// TIA Portal V17 export
// export: Created 2025-03-05T08:01:27.4239507Z, ExportSetting WithDefaults, DisplayName Totally Integrated Automation Portal, DisplayVersion V17 Update 8, DisplayName TIA Portal Openness, DisplayVersion V17 Update 8, DisplayName TIA Portal Version Control Interface, DisplayVersion V17, DisplayName SINAMICS Startdrive Advanced, DisplayVersion V17 SP2, DisplayName SINAMICS Startdrive G110M, G120, G120C, G120D, G120P, G115D, DisplayVersion V17 SP2, DisplayName SINAMICS Startdrive G130, G150, S120, S150, SINAMICS MV, S210, DisplayVersion V17 SP2, DisplayName STEP 7 Professional, DisplayVersion V17 Update 8, DisplayName SINUMERIK ONE STEP 7 Toolbox, DisplayVersion V17 Update 12, DisplayName SINUMERIK 840D sl STEP 7 Toolbox, DisplayVersion V17 Update 12, DisplayName STEP 7 Safety, DisplayVersion V17 Update 6, DisplayName WinCC Advanced, DisplayVersion V17 Update 8
FUNCTION "FC16013_METHOD_CALLS_U02_STA2_MEAS" : Void   // FC16013, LAD
{ S7_Optimized_Access := 'TRUE' }
VERSION : 0.1
// stored: AutoNumber false, IsIECCheckEnabled false, SetENOAutomatically false, UDAEnableTagReadback false
   VAR_TEMP
      AUX_WSTRING_PART_ID_STA2 : WString;
      AUX_WCHARS : Array[0..63] of WChar;
      index : Int;
      ALARM_AUX : Bool;
   END_VAR
   VAR_TEMP   // added for the SCL form of the ladder/FBD networks
      _w1 : Bool;
      _w2 : Bool;
   END_VAR
BEGIN

REGION Network 1 (SCL): TRANSFORM TO WCHARS
   FOR #index := 0 TO 63 DO
       #AUX_WCHARS[#index] := CHAR_TO_WCHAR("DB8000_PART_STATUS".UNIT_02.STATION_2.PART_A.PART_ID[#index]);
   END_FOR;
END_REGION

REGION Network 2: TRANSFORM TO WSTRING
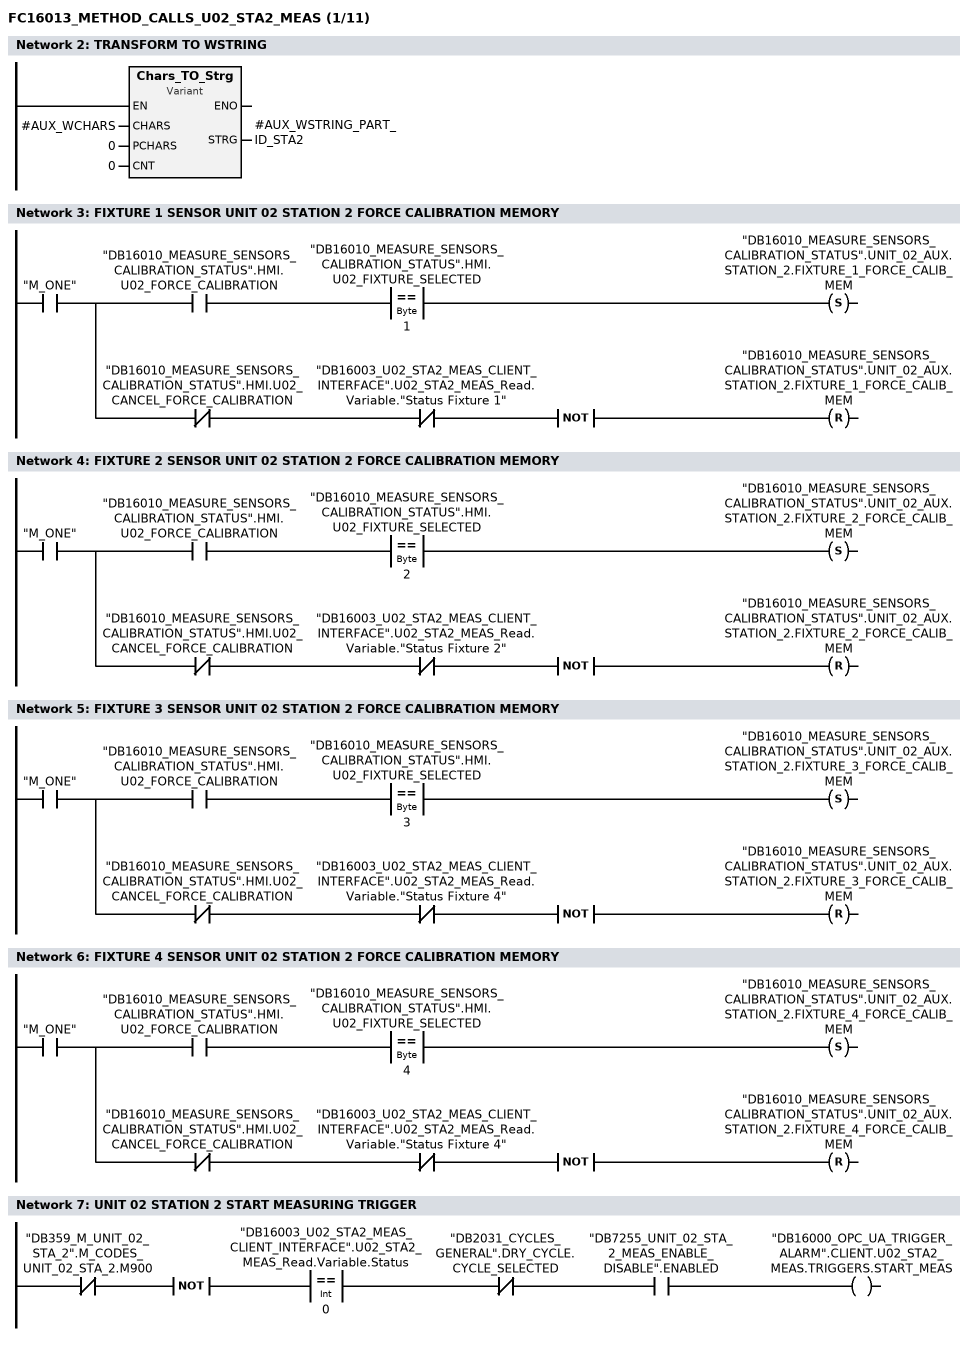
   RUNG wire#powerrail
      { S7_Templates := "[ptr_type := Variant, str_type := WString]" } Chars_TO_Strg(Chars := #AUX_WCHARS, pChars := 0, Cnt := 0, Strg => #AUX_WSTRING_PART_ID_STA2)
   END_RUNG
   // the same network as SCL:
   Chars_TO_Strg(Chars := #AUX_WCHARS, pChars := 0, Cnt := 0, Strg => #AUX_WSTRING_PART_ID_STA2);
END_REGION

REGION Network 3: FIXTURE 1 SENSOR UNIT 02 STATION 2 FORCE CALIBRATION MEMORY
   RUNG wire#powerrail
      Contact( "M_ONE" )
      wire#w1
      Contact( "DB16010_MEASURE_SENSORS_CALIBRATION_STATUS".HMI.U02_FORCE_CALIBRATION )
      { S7_Templates := "SrcType := Byte" } EQ_Contact(in1 := "DB16010_MEASURE_SENSORS_CALIBRATION_STATUS".HMI.U02_FIXTURE_SELECTED, in2 := 1)
      S_Coil( "DB16010_MEASURE_SENSORS_CALIBRATION_STATUS".UNIT_02_AUX.STATION_2.FIXTURE_1_FORCE_CALIB_MEM )
   END_RUNG
   RUNG wire#w1
      I_Contact( "DB16010_MEASURE_SENSORS_CALIBRATION_STATUS".HMI.U02_CANCEL_FORCE_CALIBRATION )
      I_Contact( "DB16003_U02_STA2_MEAS_CLIENT_INTERFACE".U02_STA2_MEAS_Read.Variable."Status Fixture 1" )
      Not()
      R_Coil( "DB16010_MEASURE_SENSORS_CALIBRATION_STATUS".UNIT_02_AUX.STATION_2.FIXTURE_1_FORCE_CALIB_MEM )
   END_RUNG
   // the same network as SCL:
   IF "M_ONE" AND "DB16010_MEASURE_SENSORS_CALIBRATION_STATUS".HMI.U02_FORCE_CALIBRATION AND ("DB16010_MEASURE_SENSORS_CALIBRATION_STATUS".HMI.U02_FIXTURE_SELECTED = 1) THEN
       "DB16010_MEASURE_SENSORS_CALIBRATION_STATUS".UNIT_02_AUX.STATION_2.FIXTURE_1_FORCE_CALIB_MEM := TRUE;
   END_IF;
   IF NOT ("M_ONE" AND NOT "DB16010_MEASURE_SENSORS_CALIBRATION_STATUS".HMI.U02_CANCEL_FORCE_CALIBRATION AND NOT "DB16003_U02_STA2_MEAS_CLIENT_INTERFACE".U02_STA2_MEAS_Read.Variable."Status Fixture 1") THEN
       "DB16010_MEASURE_SENSORS_CALIBRATION_STATUS".UNIT_02_AUX.STATION_2.FIXTURE_1_FORCE_CALIB_MEM := FALSE;
   END_IF;
END_REGION

REGION Network 4: FIXTURE 2 SENSOR UNIT 02 STATION 2 FORCE CALIBRATION MEMORY
   RUNG wire#powerrail
      Contact( "M_ONE" )
      wire#w1
      Contact( "DB16010_MEASURE_SENSORS_CALIBRATION_STATUS".HMI.U02_FORCE_CALIBRATION )
      { S7_Templates := "SrcType := Byte" } EQ_Contact(in1 := "DB16010_MEASURE_SENSORS_CALIBRATION_STATUS".HMI.U02_FIXTURE_SELECTED, in2 := 2)
      S_Coil( "DB16010_MEASURE_SENSORS_CALIBRATION_STATUS".UNIT_02_AUX.STATION_2.FIXTURE_2_FORCE_CALIB_MEM )
   END_RUNG
   RUNG wire#w1
      I_Contact( "DB16010_MEASURE_SENSORS_CALIBRATION_STATUS".HMI.U02_CANCEL_FORCE_CALIBRATION )
      I_Contact( "DB16003_U02_STA2_MEAS_CLIENT_INTERFACE".U02_STA2_MEAS_Read.Variable."Status Fixture 2" )
      Not()
      R_Coil( "DB16010_MEASURE_SENSORS_CALIBRATION_STATUS".UNIT_02_AUX.STATION_2.FIXTURE_2_FORCE_CALIB_MEM )
   END_RUNG
   // the same network as SCL:
   IF "M_ONE" AND "DB16010_MEASURE_SENSORS_CALIBRATION_STATUS".HMI.U02_FORCE_CALIBRATION AND ("DB16010_MEASURE_SENSORS_CALIBRATION_STATUS".HMI.U02_FIXTURE_SELECTED = 2) THEN
       "DB16010_MEASURE_SENSORS_CALIBRATION_STATUS".UNIT_02_AUX.STATION_2.FIXTURE_2_FORCE_CALIB_MEM := TRUE;
   END_IF;
   IF NOT ("M_ONE" AND NOT "DB16010_MEASURE_SENSORS_CALIBRATION_STATUS".HMI.U02_CANCEL_FORCE_CALIBRATION AND NOT "DB16003_U02_STA2_MEAS_CLIENT_INTERFACE".U02_STA2_MEAS_Read.Variable."Status Fixture 2") THEN
       "DB16010_MEASURE_SENSORS_CALIBRATION_STATUS".UNIT_02_AUX.STATION_2.FIXTURE_2_FORCE_CALIB_MEM := FALSE;
   END_IF;
END_REGION

REGION Network 5: FIXTURE 3 SENSOR UNIT 02 STATION 2 FORCE CALIBRATION MEMORY
   RUNG wire#powerrail
      Contact( "M_ONE" )
      wire#w1
      Contact( "DB16010_MEASURE_SENSORS_CALIBRATION_STATUS".HMI.U02_FORCE_CALIBRATION )
      { S7_Templates := "SrcType := Byte" } EQ_Contact(in1 := "DB16010_MEASURE_SENSORS_CALIBRATION_STATUS".HMI.U02_FIXTURE_SELECTED, in2 := 3)
      S_Coil( "DB16010_MEASURE_SENSORS_CALIBRATION_STATUS".UNIT_02_AUX.STATION_2.FIXTURE_3_FORCE_CALIB_MEM )
   END_RUNG
   RUNG wire#w1
      I_Contact( "DB16010_MEASURE_SENSORS_CALIBRATION_STATUS".HMI.U02_CANCEL_FORCE_CALIBRATION )
      I_Contact( "DB16003_U02_STA2_MEAS_CLIENT_INTERFACE".U02_STA2_MEAS_Read.Variable."Status Fixture 4" )
      Not()
      R_Coil( "DB16010_MEASURE_SENSORS_CALIBRATION_STATUS".UNIT_02_AUX.STATION_2.FIXTURE_3_FORCE_CALIB_MEM )
   END_RUNG
   // the same network as SCL:
   IF "M_ONE" AND "DB16010_MEASURE_SENSORS_CALIBRATION_STATUS".HMI.U02_FORCE_CALIBRATION AND ("DB16010_MEASURE_SENSORS_CALIBRATION_STATUS".HMI.U02_FIXTURE_SELECTED = 3) THEN
       "DB16010_MEASURE_SENSORS_CALIBRATION_STATUS".UNIT_02_AUX.STATION_2.FIXTURE_3_FORCE_CALIB_MEM := TRUE;
   END_IF;
   IF NOT ("M_ONE" AND NOT "DB16010_MEASURE_SENSORS_CALIBRATION_STATUS".HMI.U02_CANCEL_FORCE_CALIBRATION AND NOT "DB16003_U02_STA2_MEAS_CLIENT_INTERFACE".U02_STA2_MEAS_Read.Variable."Status Fixture 4") THEN
       "DB16010_MEASURE_SENSORS_CALIBRATION_STATUS".UNIT_02_AUX.STATION_2.FIXTURE_3_FORCE_CALIB_MEM := FALSE;
   END_IF;
END_REGION

REGION Network 6: FIXTURE 4 SENSOR UNIT 02 STATION 2 FORCE CALIBRATION MEMORY
   RUNG wire#powerrail
      Contact( "M_ONE" )
      wire#w1
      Contact( "DB16010_MEASURE_SENSORS_CALIBRATION_STATUS".HMI.U02_FORCE_CALIBRATION )
      { S7_Templates := "SrcType := Byte" } EQ_Contact(in1 := "DB16010_MEASURE_SENSORS_CALIBRATION_STATUS".HMI.U02_FIXTURE_SELECTED, in2 := 4)
      S_Coil( "DB16010_MEASURE_SENSORS_CALIBRATION_STATUS".UNIT_02_AUX.STATION_2.FIXTURE_4_FORCE_CALIB_MEM )
   END_RUNG
   RUNG wire#w1
      I_Contact( "DB16010_MEASURE_SENSORS_CALIBRATION_STATUS".HMI.U02_CANCEL_FORCE_CALIBRATION )
      I_Contact( "DB16003_U02_STA2_MEAS_CLIENT_INTERFACE".U02_STA2_MEAS_Read.Variable."Status Fixture 4" )
      Not()
      R_Coil( "DB16010_MEASURE_SENSORS_CALIBRATION_STATUS".UNIT_02_AUX.STATION_2.FIXTURE_4_FORCE_CALIB_MEM )
   END_RUNG
   // the same network as SCL:
   IF "M_ONE" AND "DB16010_MEASURE_SENSORS_CALIBRATION_STATUS".HMI.U02_FORCE_CALIBRATION AND ("DB16010_MEASURE_SENSORS_CALIBRATION_STATUS".HMI.U02_FIXTURE_SELECTED = 4) THEN
       "DB16010_MEASURE_SENSORS_CALIBRATION_STATUS".UNIT_02_AUX.STATION_2.FIXTURE_4_FORCE_CALIB_MEM := TRUE;
   END_IF;
   IF NOT ("M_ONE" AND NOT "DB16010_MEASURE_SENSORS_CALIBRATION_STATUS".HMI.U02_CANCEL_FORCE_CALIBRATION AND NOT "DB16003_U02_STA2_MEAS_CLIENT_INTERFACE".U02_STA2_MEAS_Read.Variable."Status Fixture 4") THEN
       "DB16010_MEASURE_SENSORS_CALIBRATION_STATUS".UNIT_02_AUX.STATION_2.FIXTURE_4_FORCE_CALIB_MEM := FALSE;
   END_IF;
END_REGION

REGION Network 7: UNIT 02 STATION 2 START MEASURING TRIGGER
   RUNG wire#powerrail
      I_Contact( "DB359_M_UNIT_02_STA_2".M_CODES_UNIT_02_STA_2.M900 )
      Not()
      { S7_Templates := "SrcType := Int" } EQ_Contact(in1 := "DB16003_U02_STA2_MEAS_CLIENT_INTERFACE".U02_STA2_MEAS_Read.Variable.Status, in2 := 0)
      I_Contact( "DB2031_CYCLES_GENERAL".DRY_CYCLE.CYCLE_SELECTED )
      Contact( "DB7255_UNIT_02_STA_2_MEAS_ENABLE_DISABLE".ENABLED )
      Coil( "DB16000_OPC_UA_TRIGGER_ALARM".CLIENT.U02_STA2_MEAS.TRIGGERS.START_MEAS )
   END_RUNG
   // the same network as SCL:
   "DB16000_OPC_UA_TRIGGER_ALARM".CLIENT.U02_STA2_MEAS.TRIGGERS.START_MEAS := NOT (NOT "DB359_M_UNIT_02_STA_2".M_CODES_UNIT_02_STA_2.M900) AND ("DB16003_U02_STA2_MEAS_CLIENT_INTERFACE".U02_STA2_MEAS_Read.Variable.Status = 0) AND NOT "DB2031_CYCLES_GENERAL".DRY_CYCLE.CYCLE_SELECTED AND "DB7255_UNIT_02_STA_2_MEAS_ENABLE_DISABLE".ENABLED;
END_REGION

REGION Network 8: UNIT 02 STATION 2 START CALIBRATING TRIGGER
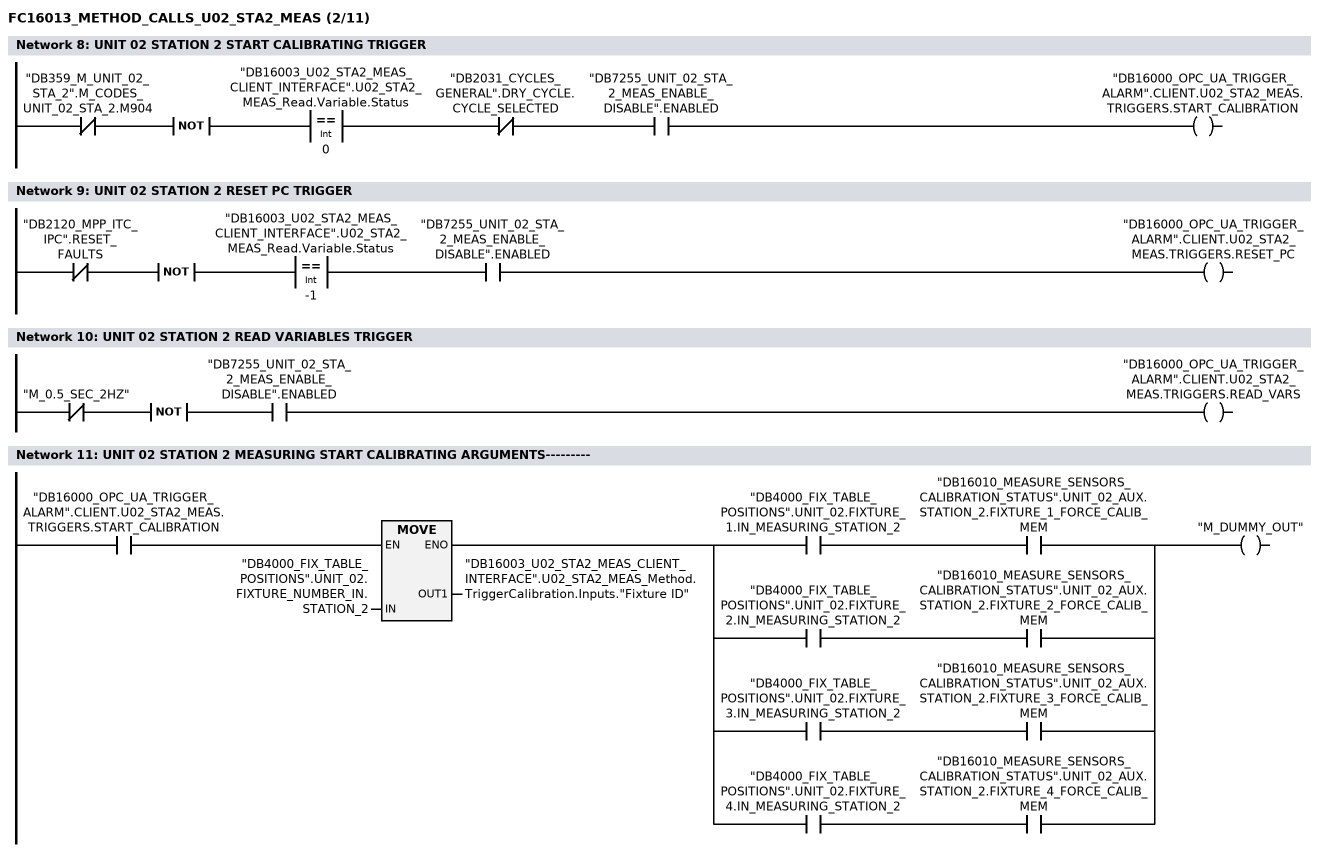
   RUNG wire#powerrail
      I_Contact( "DB359_M_UNIT_02_STA_2".M_CODES_UNIT_02_STA_2.M904 )
      Not()
      { S7_Templates := "SrcType := Int" } EQ_Contact(in1 := "DB16003_U02_STA2_MEAS_CLIENT_INTERFACE".U02_STA2_MEAS_Read.Variable.Status, in2 := 0)
      I_Contact( "DB2031_CYCLES_GENERAL".DRY_CYCLE.CYCLE_SELECTED )
      Contact( "DB7255_UNIT_02_STA_2_MEAS_ENABLE_DISABLE".ENABLED )
      Coil( "DB16000_OPC_UA_TRIGGER_ALARM".CLIENT.U02_STA2_MEAS.TRIGGERS.START_CALIBRATION )
   END_RUNG
   // the same network as SCL:
   "DB16000_OPC_UA_TRIGGER_ALARM".CLIENT.U02_STA2_MEAS.TRIGGERS.START_CALIBRATION := NOT (NOT "DB359_M_UNIT_02_STA_2".M_CODES_UNIT_02_STA_2.M904) AND ("DB16003_U02_STA2_MEAS_CLIENT_INTERFACE".U02_STA2_MEAS_Read.Variable.Status = 0) AND NOT "DB2031_CYCLES_GENERAL".DRY_CYCLE.CYCLE_SELECTED AND "DB7255_UNIT_02_STA_2_MEAS_ENABLE_DISABLE".ENABLED;
END_REGION

REGION Network 9: UNIT 02 STATION 2 RESET PC TRIGGER
   RUNG wire#powerrail
      I_Contact( "DB2120_MPP_ITC_IPC".RESET_FAULTS )
      Not()
      { S7_Templates := "SrcType := Int" } EQ_Contact(in1 := "DB16003_U02_STA2_MEAS_CLIENT_INTERFACE".U02_STA2_MEAS_Read.Variable.Status, in2 := -1)
      Contact( "DB7255_UNIT_02_STA_2_MEAS_ENABLE_DISABLE".ENABLED )
      Coil( "DB16000_OPC_UA_TRIGGER_ALARM".CLIENT.U02_STA2_MEAS.TRIGGERS.RESET_PC )
   END_RUNG
   // the same network as SCL:
   "DB16000_OPC_UA_TRIGGER_ALARM".CLIENT.U02_STA2_MEAS.TRIGGERS.RESET_PC := NOT (NOT "DB2120_MPP_ITC_IPC".RESET_FAULTS) AND ("DB16003_U02_STA2_MEAS_CLIENT_INTERFACE".U02_STA2_MEAS_Read.Variable.Status = (-1)) AND "DB7255_UNIT_02_STA_2_MEAS_ENABLE_DISABLE".ENABLED;
END_REGION

REGION Network 10: UNIT 02 STATION 2 READ VARIABLES TRIGGER
   RUNG wire#powerrail
      I_Contact( "M_0.5_SEC_2HZ" )
      Not()
      Contact( "DB7255_UNIT_02_STA_2_MEAS_ENABLE_DISABLE".ENABLED )
      Coil( "DB16000_OPC_UA_TRIGGER_ALARM".CLIENT.U02_STA2_MEAS.TRIGGERS.READ_VARS )
   END_RUNG
   // the same network as SCL:
   "DB16000_OPC_UA_TRIGGER_ALARM".CLIENT.U02_STA2_MEAS.TRIGGERS.READ_VARS := NOT (NOT "M_0.5_SEC_2HZ") AND "DB7255_UNIT_02_STA_2_MEAS_ENABLE_DISABLE".ENABLED;
END_REGION

REGION Network 11: UNIT 02 STATION 2 MEASURING START CALIBRATING ARGUMENTS---------
   RUNG wire#powerrail
      Contact( "DB16000_OPC_UA_TRIGGER_ALARM".CLIENT.U02_STA2_MEAS.TRIGGERS.START_CALIBRATION )
      Move(in := "DB4000_FIX_TABLE_POSITIONS".UNIT_02.FIXTURE_NUMBER_IN.STATION_2, out1 => "DB16003_U02_STA2_MEAS_CLIENT_INTERFACE".U02_STA2_MEAS_Method.TriggerCalibration.Inputs."Fixture ID")
      wire#w1
      Contact( "DB4000_FIX_TABLE_POSITIONS".UNIT_02.FIXTURE_1.IN_MEASURING_STATION_2 )
      Contact( "DB16010_MEASURE_SENSORS_CALIBRATION_STATUS".UNIT_02_AUX.STATION_2.FIXTURE_1_FORCE_CALIB_MEM )
      wire#w2
      Coil( "M_DUMMY_OUT" )
   END_RUNG
   RUNG wire#w1
      Contact( "DB4000_FIX_TABLE_POSITIONS".UNIT_02.FIXTURE_2.IN_MEASURING_STATION_2 )
      Contact( "DB16010_MEASURE_SENSORS_CALIBRATION_STATUS".UNIT_02_AUX.STATION_2.FIXTURE_2_FORCE_CALIB_MEM )
   END_RUNG wire#w2
   RUNG wire#w1
      Contact( "DB4000_FIX_TABLE_POSITIONS".UNIT_02.FIXTURE_3.IN_MEASURING_STATION_2 )
      Contact( "DB16010_MEASURE_SENSORS_CALIBRATION_STATUS".UNIT_02_AUX.STATION_2.FIXTURE_3_FORCE_CALIB_MEM )
   END_RUNG wire#w2
   RUNG wire#w1
      Contact( "DB4000_FIX_TABLE_POSITIONS".UNIT_02.FIXTURE_4.IN_MEASURING_STATION_2 )
      Contact( "DB16010_MEASURE_SENSORS_CALIBRATION_STATUS".UNIT_02_AUX.STATION_2.FIXTURE_4_FORCE_CALIB_MEM )
   END_RUNG wire#w2
   // the same network as SCL:
   IF "DB16000_OPC_UA_TRIGGER_ALARM".CLIENT.U02_STA2_MEAS.TRIGGERS.START_CALIBRATION THEN
       "DB16003_U02_STA2_MEAS_CLIENT_INTERFACE".U02_STA2_MEAS_Method.TriggerCalibration.Inputs."Fixture ID" := "DB4000_FIX_TABLE_POSITIONS".UNIT_02.FIXTURE_NUMBER_IN.STATION_2;
   END_IF;
   "M_DUMMY_OUT" := "DB16000_OPC_UA_TRIGGER_ALARM".CLIENT.U02_STA2_MEAS.TRIGGERS.START_CALIBRATION AND (("DB4000_FIX_TABLE_POSITIONS".UNIT_02.FIXTURE_1.IN_MEASURING_STATION_2 AND "DB16010_MEASURE_SENSORS_CALIBRATION_STATUS".UNIT_02_AUX.STATION_2.FIXTURE_1_FORCE_CALIB_MEM) OR ("DB4000_FIX_TABLE_POSITIONS".UNIT_02.FIXTURE_2.IN_MEASURING_STATION_2 AND "DB16010_MEASURE_SENSORS_CALIBRATION_STATUS".UNIT_02_AUX.STATION_2.FIXTURE_2_FORCE_CALIB_MEM) OR ("DB4000_FIX_TABLE_POSITIONS".UNIT_02.FIXTURE_3.IN_MEASURING_STATION_2 AND "DB16010_MEASURE_SENSORS_CALIBRATION_STATUS".UNIT_02_AUX.STATION_2.FIXTURE_3_FORCE_CALIB_MEM) OR ("DB4000_FIX_TABLE_POSITIONS".UNIT_02.FIXTURE_4.IN_MEASURING_STATION_2 AND "DB16010_MEASURE_SENSORS_CALIBRATION_STATUS".UNIT_02_AUX.STATION_2.FIXTURE_4_FORCE_CALIB_MEM));
END_REGION

REGION Network 12: UNIT 02 STATION 2 START MEASURING TRIGGER CALL
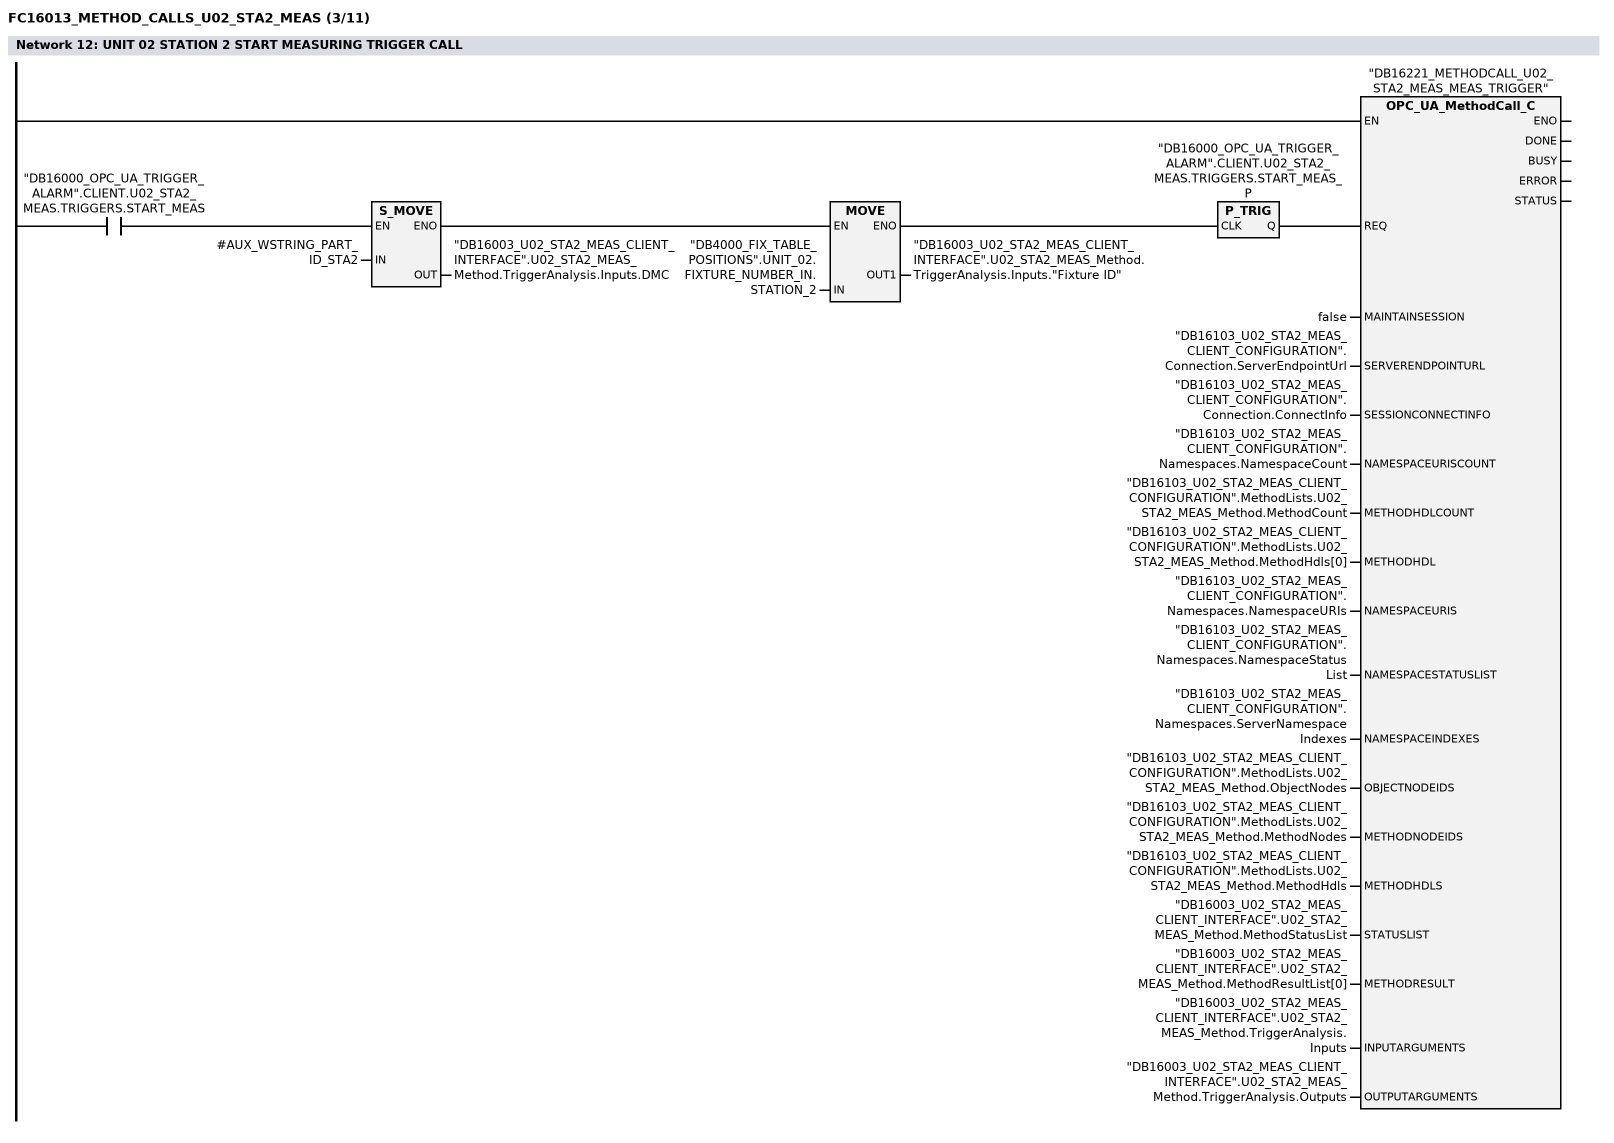
   RUNG wire#powerrail
      "DB16221_METHODCALL_U02_STA2_MEAS_MEAS_TRIGGER".OPC_UA_MethodCall_C(REQ := wire#w1, MaintainSession := false, ServerEndpointUrl := "DB16103_U02_STA2_MEAS_CLIENT_CONFIGURATION".Connection.ServerEndpointUrl, SessionConnectInfo := "DB16103_U02_STA2_MEAS_CLIENT_CONFIGURATION".Connection.ConnectInfo, NamespaceUrisCount := "DB16103_U02_STA2_MEAS_CLIENT_CONFIGURATION".Namespaces.NamespaceCount, MethodHdlCount := "DB16103_U02_STA2_MEAS_CLIENT_CONFIGURATION".MethodLists.U02_STA2_MEAS_Method.MethodCount, MethodHdl := "DB16103_U02_STA2_MEAS_CLIENT_CONFIGURATION".MethodLists.U02_STA2_MEAS_Method.MethodHdls[0], NamespaceUris := "DB16103_U02_STA2_MEAS_CLIENT_CONFIGURATION".Namespaces.NamespaceURIs, NamespaceStatusList := "DB16103_U02_STA2_MEAS_CLIENT_CONFIGURATION".Namespaces.NamespaceStatusList, NamespaceIndexes := "DB16103_U02_STA2_MEAS_CLIENT_CONFIGURATION".Namespaces.ServerNamespaceIndexes, ObjectNodeIDs := "DB16103_U02_STA2_MEAS_CLIENT_CONFIGURATION".MethodLists.U02_STA2_MEAS_Method.ObjectNodes, MethodNodeIDs := "DB16103_U02_STA2_MEAS_CLIENT_CONFIGURATION".MethodLists.U02_STA2_MEAS_Method.MethodNodes, MethodHdls := "DB16103_U02_STA2_MEAS_CLIENT_CONFIGURATION".MethodLists.U02_STA2_MEAS_Method.MethodHdls, StatusList := "DB16003_U02_STA2_MEAS_CLIENT_INTERFACE".U02_STA2_MEAS_Method.MethodStatusList, MethodResult := "DB16003_U02_STA2_MEAS_CLIENT_INTERFACE".U02_STA2_MEAS_Method.MethodResultList[0], InputArguments := "DB16003_U02_STA2_MEAS_CLIENT_INTERFACE".U02_STA2_MEAS_Method.TriggerAnalysis.Inputs, OutputArguments := "DB16003_U02_STA2_MEAS_CLIENT_INTERFACE".U02_STA2_MEAS_Method.TriggerAnalysis.Outputs, Done =>, Busy =>, Error =>, Status =>)
   END_RUNG
   RUNG wire#powerrail
      Contact( "DB16000_OPC_UA_TRIGGER_ALARM".CLIENT.U02_STA2_MEAS.TRIGGERS.START_MEAS )
      S_Move(in := #AUX_WSTRING_PART_ID_STA2, out => "DB16003_U02_STA2_MEAS_CLIENT_INTERFACE".U02_STA2_MEAS_Method.TriggerAnalysis.Inputs.DMC)
      Move(in := "DB4000_FIX_TABLE_POSITIONS".UNIT_02.FIXTURE_NUMBER_IN.STATION_2, out1 => "DB16003_U02_STA2_MEAS_CLIENT_INTERFACE".U02_STA2_MEAS_Method.TriggerAnalysis.Inputs."Fixture ID")
      P_Trig( "DB16000_OPC_UA_TRIGGER_ALARM".CLIENT.U02_STA2_MEAS.TRIGGERS.START_MEAS_P )
   END_RUNG wire#w1
   // the same network as SCL:
   IF "DB16000_OPC_UA_TRIGGER_ALARM".CLIENT.U02_STA2_MEAS.TRIGGERS.START_MEAS THEN
       "DB16003_U02_STA2_MEAS_CLIENT_INTERFACE".U02_STA2_MEAS_Method.TriggerAnalysis.Inputs.DMC := #AUX_WSTRING_PART_ID_STA2;
       "DB16003_U02_STA2_MEAS_CLIENT_INTERFACE".U02_STA2_MEAS_Method.TriggerAnalysis.Inputs."Fixture ID" := "DB4000_FIX_TABLE_POSITIONS".UNIT_02.FIXTURE_NUMBER_IN.STATION_2;
   END_IF;
   #_w1 := "DB16000_OPC_UA_TRIGGER_ALARM".CLIENT.U02_STA2_MEAS.TRIGGERS.START_MEAS AND NOT "DB16000_OPC_UA_TRIGGER_ALARM".CLIENT.U02_STA2_MEAS.TRIGGERS.START_MEAS_P;   // rising edge
   "DB16000_OPC_UA_TRIGGER_ALARM".CLIENT.U02_STA2_MEAS.TRIGGERS.START_MEAS_P := "DB16000_OPC_UA_TRIGGER_ALARM".CLIENT.U02_STA2_MEAS.TRIGGERS.START_MEAS;
   "DB16221_METHODCALL_U02_STA2_MEAS_MEAS_TRIGGER"(REQ := #_w1,   // OPC_UA_MethodCall_C
                           MaintainSession := false,
                           ServerEndpointUrl := "DB16103_U02_STA2_MEAS_CLIENT_CONFIGURATION".Connection.ServerEndpointUrl,
                           SessionConnectInfo := "DB16103_U02_STA2_MEAS_CLIENT_CONFIGURATION".Connection.ConnectInfo,
                           NamespaceUrisCount := "DB16103_U02_STA2_MEAS_CLIENT_CONFIGURATION".Namespaces.NamespaceCount,
                           MethodHdlCount := "DB16103_U02_STA2_MEAS_CLIENT_CONFIGURATION".MethodLists.U02_STA2_MEAS_Method.MethodCount,
                           MethodHdl := "DB16103_U02_STA2_MEAS_CLIENT_CONFIGURATION".MethodLists.U02_STA2_MEAS_Method.MethodHdls[0],
                           NamespaceUris := "DB16103_U02_STA2_MEAS_CLIENT_CONFIGURATION".Namespaces.NamespaceURIs,
                           NamespaceStatusList := "DB16103_U02_STA2_MEAS_CLIENT_CONFIGURATION".Namespaces.NamespaceStatusList,
                           NamespaceIndexes := "DB16103_U02_STA2_MEAS_CLIENT_CONFIGURATION".Namespaces.ServerNamespaceIndexes,
                           ObjectNodeIDs := "DB16103_U02_STA2_MEAS_CLIENT_CONFIGURATION".MethodLists.U02_STA2_MEAS_Method.ObjectNodes,
                           MethodNodeIDs := "DB16103_U02_STA2_MEAS_CLIENT_CONFIGURATION".MethodLists.U02_STA2_MEAS_Method.MethodNodes,
                           MethodHdls := "DB16103_U02_STA2_MEAS_CLIENT_CONFIGURATION".MethodLists.U02_STA2_MEAS_Method.MethodHdls,
                           StatusList := "DB16003_U02_STA2_MEAS_CLIENT_INTERFACE".U02_STA2_MEAS_Method.MethodStatusList,
                           MethodResult := "DB16003_U02_STA2_MEAS_CLIENT_INTERFACE".U02_STA2_MEAS_Method.MethodResultList[0],
                           InputArguments := "DB16003_U02_STA2_MEAS_CLIENT_INTERFACE".U02_STA2_MEAS_Method.TriggerAnalysis.Inputs,
                           OutputArguments := "DB16003_U02_STA2_MEAS_CLIENT_INTERFACE".U02_STA2_MEAS_Method.TriggerAnalysis.Outputs);
END_REGION

REGION Network 13: UNIT 02 STATION 2 START CALIBRATING TRIGGER CALL
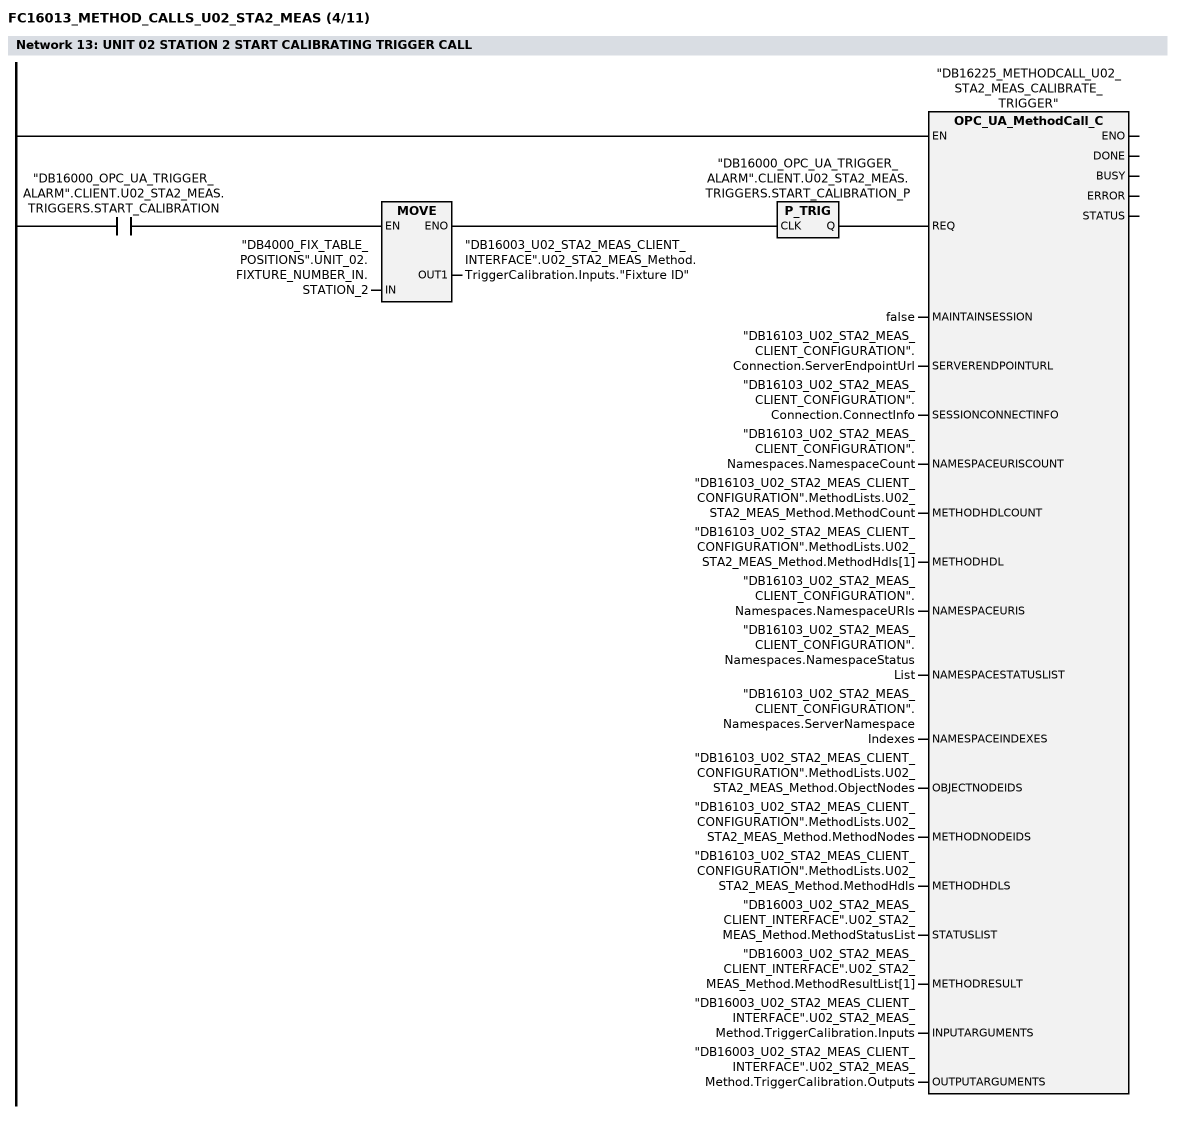
   RUNG wire#powerrail
      "DB16225_METHODCALL_U02_STA2_MEAS_CALIBRATE_TRIGGER".OPC_UA_MethodCall_C(REQ := wire#w1, MaintainSession := false, ServerEndpointUrl := "DB16103_U02_STA2_MEAS_CLIENT_CONFIGURATION".Connection.ServerEndpointUrl, SessionConnectInfo := "DB16103_U02_STA2_MEAS_CLIENT_CONFIGURATION".Connection.ConnectInfo, NamespaceUrisCount := "DB16103_U02_STA2_MEAS_CLIENT_CONFIGURATION".Namespaces.NamespaceCount, MethodHdlCount := "DB16103_U02_STA2_MEAS_CLIENT_CONFIGURATION".MethodLists.U02_STA2_MEAS_Method.MethodCount, MethodHdl := "DB16103_U02_STA2_MEAS_CLIENT_CONFIGURATION".MethodLists.U02_STA2_MEAS_Method.MethodHdls[1], NamespaceUris := "DB16103_U02_STA2_MEAS_CLIENT_CONFIGURATION".Namespaces.NamespaceURIs, NamespaceStatusList := "DB16103_U02_STA2_MEAS_CLIENT_CONFIGURATION".Namespaces.NamespaceStatusList, NamespaceIndexes := "DB16103_U02_STA2_MEAS_CLIENT_CONFIGURATION".Namespaces.ServerNamespaceIndexes, ObjectNodeIDs := "DB16103_U02_STA2_MEAS_CLIENT_CONFIGURATION".MethodLists.U02_STA2_MEAS_Method.ObjectNodes, MethodNodeIDs := "DB16103_U02_STA2_MEAS_CLIENT_CONFIGURATION".MethodLists.U02_STA2_MEAS_Method.MethodNodes, MethodHdls := "DB16103_U02_STA2_MEAS_CLIENT_CONFIGURATION".MethodLists.U02_STA2_MEAS_Method.MethodHdls, StatusList := "DB16003_U02_STA2_MEAS_CLIENT_INTERFACE".U02_STA2_MEAS_Method.MethodStatusList, MethodResult := "DB16003_U02_STA2_MEAS_CLIENT_INTERFACE".U02_STA2_MEAS_Method.MethodResultList[1], InputArguments := "DB16003_U02_STA2_MEAS_CLIENT_INTERFACE".U02_STA2_MEAS_Method.TriggerCalibration.Inputs, OutputArguments := "DB16003_U02_STA2_MEAS_CLIENT_INTERFACE".U02_STA2_MEAS_Method.TriggerCalibration.Outputs, Done =>, Busy =>, Error =>, Status =>)
   END_RUNG
   RUNG wire#powerrail
      Contact( "DB16000_OPC_UA_TRIGGER_ALARM".CLIENT.U02_STA2_MEAS.TRIGGERS.START_CALIBRATION )
      Move(in := "DB4000_FIX_TABLE_POSITIONS".UNIT_02.FIXTURE_NUMBER_IN.STATION_2, out1 => "DB16003_U02_STA2_MEAS_CLIENT_INTERFACE".U02_STA2_MEAS_Method.TriggerCalibration.Inputs."Fixture ID")
      P_Trig( "DB16000_OPC_UA_TRIGGER_ALARM".CLIENT.U02_STA2_MEAS.TRIGGERS.START_CALIBRATION_P )
   END_RUNG wire#w1
   // the same network as SCL:
   IF "DB16000_OPC_UA_TRIGGER_ALARM".CLIENT.U02_STA2_MEAS.TRIGGERS.START_CALIBRATION THEN
       "DB16003_U02_STA2_MEAS_CLIENT_INTERFACE".U02_STA2_MEAS_Method.TriggerCalibration.Inputs."Fixture ID" := "DB4000_FIX_TABLE_POSITIONS".UNIT_02.FIXTURE_NUMBER_IN.STATION_2;
   END_IF;
   #_w1 := "DB16000_OPC_UA_TRIGGER_ALARM".CLIENT.U02_STA2_MEAS.TRIGGERS.START_CALIBRATION AND NOT "DB16000_OPC_UA_TRIGGER_ALARM".CLIENT.U02_STA2_MEAS.TRIGGERS.START_CALIBRATION_P;   // rising edge
   "DB16000_OPC_UA_TRIGGER_ALARM".CLIENT.U02_STA2_MEAS.TRIGGERS.START_CALIBRATION_P := "DB16000_OPC_UA_TRIGGER_ALARM".CLIENT.U02_STA2_MEAS.TRIGGERS.START_CALIBRATION;
   "DB16225_METHODCALL_U02_STA2_MEAS_CALIBRATE_TRIGGER"(REQ := #_w1,   // OPC_UA_MethodCall_C
                           MaintainSession := false,
                           ServerEndpointUrl := "DB16103_U02_STA2_MEAS_CLIENT_CONFIGURATION".Connection.ServerEndpointUrl,
                           SessionConnectInfo := "DB16103_U02_STA2_MEAS_CLIENT_CONFIGURATION".Connection.ConnectInfo,
                           NamespaceUrisCount := "DB16103_U02_STA2_MEAS_CLIENT_CONFIGURATION".Namespaces.NamespaceCount,
                           MethodHdlCount := "DB16103_U02_STA2_MEAS_CLIENT_CONFIGURATION".MethodLists.U02_STA2_MEAS_Method.MethodCount,
                           MethodHdl := "DB16103_U02_STA2_MEAS_CLIENT_CONFIGURATION".MethodLists.U02_STA2_MEAS_Method.MethodHdls[1],
                           NamespaceUris := "DB16103_U02_STA2_MEAS_CLIENT_CONFIGURATION".Namespaces.NamespaceURIs,
                           NamespaceStatusList := "DB16103_U02_STA2_MEAS_CLIENT_CONFIGURATION".Namespaces.NamespaceStatusList,
                           NamespaceIndexes := "DB16103_U02_STA2_MEAS_CLIENT_CONFIGURATION".Namespaces.ServerNamespaceIndexes,
                           ObjectNodeIDs := "DB16103_U02_STA2_MEAS_CLIENT_CONFIGURATION".MethodLists.U02_STA2_MEAS_Method.ObjectNodes,
                           MethodNodeIDs := "DB16103_U02_STA2_MEAS_CLIENT_CONFIGURATION".MethodLists.U02_STA2_MEAS_Method.MethodNodes,
                           MethodHdls := "DB16103_U02_STA2_MEAS_CLIENT_CONFIGURATION".MethodLists.U02_STA2_MEAS_Method.MethodHdls,
                           StatusList := "DB16003_U02_STA2_MEAS_CLIENT_INTERFACE".U02_STA2_MEAS_Method.MethodStatusList,
                           MethodResult := "DB16003_U02_STA2_MEAS_CLIENT_INTERFACE".U02_STA2_MEAS_Method.MethodResultList[1],
                           InputArguments := "DB16003_U02_STA2_MEAS_CLIENT_INTERFACE".U02_STA2_MEAS_Method.TriggerCalibration.Inputs,
                           OutputArguments := "DB16003_U02_STA2_MEAS_CLIENT_INTERFACE".U02_STA2_MEAS_Method.TriggerCalibration.Outputs);
END_REGION

REGION Network 14: UNIT 02 STATION 2 RESET PC TRIGGER CALL
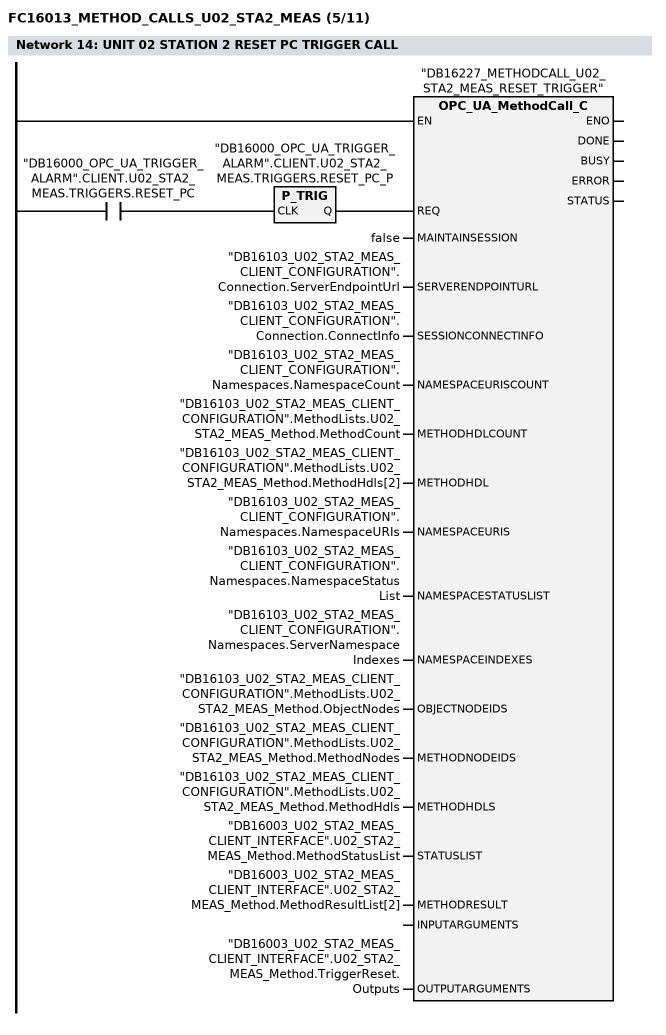
   RUNG wire#powerrail
      "DB16227_METHODCALL_U02_STA2_MEAS_RESET_TRIGGER".OPC_UA_MethodCall_C(REQ := wire#w1, MaintainSession := false, ServerEndpointUrl := "DB16103_U02_STA2_MEAS_CLIENT_CONFIGURATION".Connection.ServerEndpointUrl, SessionConnectInfo := "DB16103_U02_STA2_MEAS_CLIENT_CONFIGURATION".Connection.ConnectInfo, NamespaceUrisCount := "DB16103_U02_STA2_MEAS_CLIENT_CONFIGURATION".Namespaces.NamespaceCount, MethodHdlCount := "DB16103_U02_STA2_MEAS_CLIENT_CONFIGURATION".MethodLists.U02_STA2_MEAS_Method.MethodCount, MethodHdl := "DB16103_U02_STA2_MEAS_CLIENT_CONFIGURATION".MethodLists.U02_STA2_MEAS_Method.MethodHdls[2], NamespaceUris := "DB16103_U02_STA2_MEAS_CLIENT_CONFIGURATION".Namespaces.NamespaceURIs, NamespaceStatusList := "DB16103_U02_STA2_MEAS_CLIENT_CONFIGURATION".Namespaces.NamespaceStatusList, NamespaceIndexes := "DB16103_U02_STA2_MEAS_CLIENT_CONFIGURATION".Namespaces.ServerNamespaceIndexes, ObjectNodeIDs := "DB16103_U02_STA2_MEAS_CLIENT_CONFIGURATION".MethodLists.U02_STA2_MEAS_Method.ObjectNodes, MethodNodeIDs := "DB16103_U02_STA2_MEAS_CLIENT_CONFIGURATION".MethodLists.U02_STA2_MEAS_Method.MethodNodes, MethodHdls := "DB16103_U02_STA2_MEAS_CLIENT_CONFIGURATION".MethodLists.U02_STA2_MEAS_Method.MethodHdls, StatusList := "DB16003_U02_STA2_MEAS_CLIENT_INTERFACE".U02_STA2_MEAS_Method.MethodStatusList, MethodResult := "DB16003_U02_STA2_MEAS_CLIENT_INTERFACE".U02_STA2_MEAS_Method.MethodResultList[2], InputArguments :=, OutputArguments := "DB16003_U02_STA2_MEAS_CLIENT_INTERFACE".U02_STA2_MEAS_Method.TriggerReset.Outputs, Done =>, Busy =>, Error =>, Status =>)
   END_RUNG
   RUNG wire#powerrail
      Contact( "DB16000_OPC_UA_TRIGGER_ALARM".CLIENT.U02_STA2_MEAS.TRIGGERS.RESET_PC )
      P_Trig( "DB16000_OPC_UA_TRIGGER_ALARM".CLIENT.U02_STA2_MEAS.TRIGGERS.RESET_PC_P )
   END_RUNG wire#w1
   // the same network as SCL:
   #_w1 := "DB16000_OPC_UA_TRIGGER_ALARM".CLIENT.U02_STA2_MEAS.TRIGGERS.RESET_PC AND NOT "DB16000_OPC_UA_TRIGGER_ALARM".CLIENT.U02_STA2_MEAS.TRIGGERS.RESET_PC_P;   // rising edge
   "DB16000_OPC_UA_TRIGGER_ALARM".CLIENT.U02_STA2_MEAS.TRIGGERS.RESET_PC_P := "DB16000_OPC_UA_TRIGGER_ALARM".CLIENT.U02_STA2_MEAS.TRIGGERS.RESET_PC;
   "DB16227_METHODCALL_U02_STA2_MEAS_RESET_TRIGGER"(REQ := #_w1,   // OPC_UA_MethodCall_C
                           MaintainSession := false,
                           ServerEndpointUrl := "DB16103_U02_STA2_MEAS_CLIENT_CONFIGURATION".Connection.ServerEndpointUrl,
                           SessionConnectInfo := "DB16103_U02_STA2_MEAS_CLIENT_CONFIGURATION".Connection.ConnectInfo,
                           NamespaceUrisCount := "DB16103_U02_STA2_MEAS_CLIENT_CONFIGURATION".Namespaces.NamespaceCount,
                           MethodHdlCount := "DB16103_U02_STA2_MEAS_CLIENT_CONFIGURATION".MethodLists.U02_STA2_MEAS_Method.MethodCount,
                           MethodHdl := "DB16103_U02_STA2_MEAS_CLIENT_CONFIGURATION".MethodLists.U02_STA2_MEAS_Method.MethodHdls[2],
                           NamespaceUris := "DB16103_U02_STA2_MEAS_CLIENT_CONFIGURATION".Namespaces.NamespaceURIs,
                           NamespaceStatusList := "DB16103_U02_STA2_MEAS_CLIENT_CONFIGURATION".Namespaces.NamespaceStatusList,
                           NamespaceIndexes := "DB16103_U02_STA2_MEAS_CLIENT_CONFIGURATION".Namespaces.ServerNamespaceIndexes,
                           ObjectNodeIDs := "DB16103_U02_STA2_MEAS_CLIENT_CONFIGURATION".MethodLists.U02_STA2_MEAS_Method.ObjectNodes,
                           MethodNodeIDs := "DB16103_U02_STA2_MEAS_CLIENT_CONFIGURATION".MethodLists.U02_STA2_MEAS_Method.MethodNodes,
                           MethodHdls := "DB16103_U02_STA2_MEAS_CLIENT_CONFIGURATION".MethodLists.U02_STA2_MEAS_Method.MethodHdls,
                           StatusList := "DB16003_U02_STA2_MEAS_CLIENT_INTERFACE".U02_STA2_MEAS_Method.MethodStatusList,
                           MethodResult := "DB16003_U02_STA2_MEAS_CLIENT_INTERFACE".U02_STA2_MEAS_Method.MethodResultList[2],
                           OutputArguments := "DB16003_U02_STA2_MEAS_CLIENT_INTERFACE".U02_STA2_MEAS_Method.TriggerReset.Outputs);
END_REGION

REGION Network 15: UNIT 02 STATION 2 READ VARIABLES TRIGGER CALL
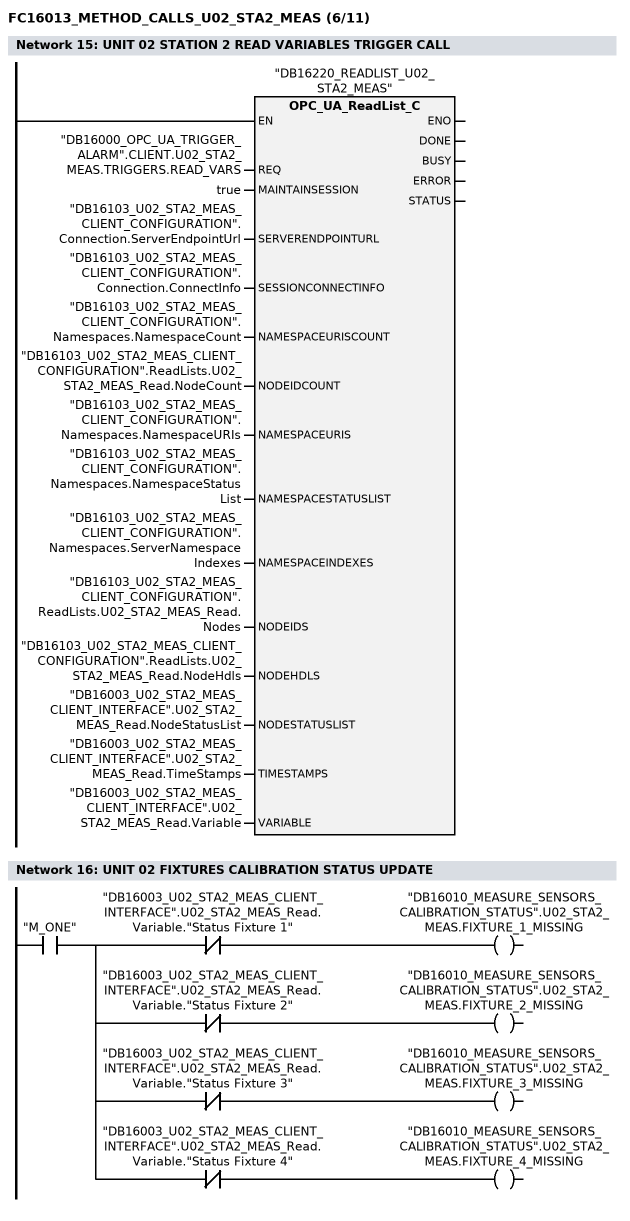
   RUNG wire#powerrail
      "DB16220_READLIST_U02_STA2_MEAS".OPC_UA_ReadList_C(REQ := "DB16000_OPC_UA_TRIGGER_ALARM".CLIENT.U02_STA2_MEAS.TRIGGERS.READ_VARS, MaintainSession := true, ServerEndpointUrl := "DB16103_U02_STA2_MEAS_CLIENT_CONFIGURATION".Connection.ServerEndpointUrl, SessionConnectInfo := "DB16103_U02_STA2_MEAS_CLIENT_CONFIGURATION".Connection.ConnectInfo, NamespaceUrisCount := "DB16103_U02_STA2_MEAS_CLIENT_CONFIGURATION".Namespaces.NamespaceCount, NodeIDCount := "DB16103_U02_STA2_MEAS_CLIENT_CONFIGURATION".ReadLists.U02_STA2_MEAS_Read.NodeCount, NamespaceUris := "DB16103_U02_STA2_MEAS_CLIENT_CONFIGURATION".Namespaces.NamespaceURIs, NamespaceStatusList := "DB16103_U02_STA2_MEAS_CLIENT_CONFIGURATION".Namespaces.NamespaceStatusList, NamespaceIndexes := "DB16103_U02_STA2_MEAS_CLIENT_CONFIGURATION".Namespaces.ServerNamespaceIndexes, NodeIDs := "DB16103_U02_STA2_MEAS_CLIENT_CONFIGURATION".ReadLists.U02_STA2_MEAS_Read.Nodes, NodeHdls := "DB16103_U02_STA2_MEAS_CLIENT_CONFIGURATION".ReadLists.U02_STA2_MEAS_Read.NodeHdls, NodeStatusList := "DB16003_U02_STA2_MEAS_CLIENT_INTERFACE".U02_STA2_MEAS_Read.NodeStatusList, Timestamps := "DB16003_U02_STA2_MEAS_CLIENT_INTERFACE".U02_STA2_MEAS_Read.TimeStamps, Variable := "DB16003_U02_STA2_MEAS_CLIENT_INTERFACE".U02_STA2_MEAS_Read.Variable, Done =>, Busy =>, Error =>, Status =>)
   END_RUNG
   // the same network as SCL:
   "DB16220_READLIST_U02_STA2_MEAS"(REQ := "DB16000_OPC_UA_TRIGGER_ALARM".CLIENT.U02_STA2_MEAS.TRIGGERS.READ_VARS,   // OPC_UA_ReadList_C
                           MaintainSession := true,
                           ServerEndpointUrl := "DB16103_U02_STA2_MEAS_CLIENT_CONFIGURATION".Connection.ServerEndpointUrl,
                           SessionConnectInfo := "DB16103_U02_STA2_MEAS_CLIENT_CONFIGURATION".Connection.ConnectInfo,
                           NamespaceUrisCount := "DB16103_U02_STA2_MEAS_CLIENT_CONFIGURATION".Namespaces.NamespaceCount,
                           NodeIDCount := "DB16103_U02_STA2_MEAS_CLIENT_CONFIGURATION".ReadLists.U02_STA2_MEAS_Read.NodeCount,
                           NamespaceUris := "DB16103_U02_STA2_MEAS_CLIENT_CONFIGURATION".Namespaces.NamespaceURIs,
                           NamespaceStatusList := "DB16103_U02_STA2_MEAS_CLIENT_CONFIGURATION".Namespaces.NamespaceStatusList,
                           NamespaceIndexes := "DB16103_U02_STA2_MEAS_CLIENT_CONFIGURATION".Namespaces.ServerNamespaceIndexes,
                           NodeIDs := "DB16103_U02_STA2_MEAS_CLIENT_CONFIGURATION".ReadLists.U02_STA2_MEAS_Read.Nodes,
                           NodeHdls := "DB16103_U02_STA2_MEAS_CLIENT_CONFIGURATION".ReadLists.U02_STA2_MEAS_Read.NodeHdls,
                           NodeStatusList := "DB16003_U02_STA2_MEAS_CLIENT_INTERFACE".U02_STA2_MEAS_Read.NodeStatusList,
                           Timestamps := "DB16003_U02_STA2_MEAS_CLIENT_INTERFACE".U02_STA2_MEAS_Read.TimeStamps,
                           Variable := "DB16003_U02_STA2_MEAS_CLIENT_INTERFACE".U02_STA2_MEAS_Read.Variable);
END_REGION

REGION Network 16: UNIT 02 FIXTURES CALIBRATION STATUS UPDATE
   RUNG wire#powerrail
      Contact( "M_ONE" )
      wire#w1
      I_Contact( "DB16003_U02_STA2_MEAS_CLIENT_INTERFACE".U02_STA2_MEAS_Read.Variable."Status Fixture 1" )
      Coil( "DB16010_MEASURE_SENSORS_CALIBRATION_STATUS".U02_STA2_MEAS.FIXTURE_1_MISSING )
   END_RUNG
   RUNG wire#w1
      I_Contact( "DB16003_U02_STA2_MEAS_CLIENT_INTERFACE".U02_STA2_MEAS_Read.Variable."Status Fixture 2" )
      Coil( "DB16010_MEASURE_SENSORS_CALIBRATION_STATUS".U02_STA2_MEAS.FIXTURE_2_MISSING )
   END_RUNG
   RUNG wire#w1
      I_Contact( "DB16003_U02_STA2_MEAS_CLIENT_INTERFACE".U02_STA2_MEAS_Read.Variable."Status Fixture 3" )
      Coil( "DB16010_MEASURE_SENSORS_CALIBRATION_STATUS".U02_STA2_MEAS.FIXTURE_3_MISSING )
   END_RUNG
   RUNG wire#w1
      I_Contact( "DB16003_U02_STA2_MEAS_CLIENT_INTERFACE".U02_STA2_MEAS_Read.Variable."Status Fixture 4" )
      Coil( "DB16010_MEASURE_SENSORS_CALIBRATION_STATUS".U02_STA2_MEAS.FIXTURE_4_MISSING )
   END_RUNG
   // the same network as SCL:
   "DB16010_MEASURE_SENSORS_CALIBRATION_STATUS".U02_STA2_MEAS.FIXTURE_1_MISSING := "M_ONE" AND NOT "DB16003_U02_STA2_MEAS_CLIENT_INTERFACE".U02_STA2_MEAS_Read.Variable."Status Fixture 1";
   "DB16010_MEASURE_SENSORS_CALIBRATION_STATUS".U02_STA2_MEAS.FIXTURE_2_MISSING := "M_ONE" AND NOT "DB16003_U02_STA2_MEAS_CLIENT_INTERFACE".U02_STA2_MEAS_Read.Variable."Status Fixture 2";
   "DB16010_MEASURE_SENSORS_CALIBRATION_STATUS".U02_STA2_MEAS.FIXTURE_3_MISSING := "M_ONE" AND NOT "DB16003_U02_STA2_MEAS_CLIENT_INTERFACE".U02_STA2_MEAS_Read.Variable."Status Fixture 3";
   "DB16010_MEASURE_SENSORS_CALIBRATION_STATUS".U02_STA2_MEAS.FIXTURE_4_MISSING := "M_ONE" AND NOT "DB16003_U02_STA2_MEAS_CLIENT_INTERFACE".U02_STA2_MEAS_Read.Variable."Status Fixture 4";
END_REGION

REGION Network 17: UNIT 02 STATION 2 MEASURING METHOD CONNECTION ALARM
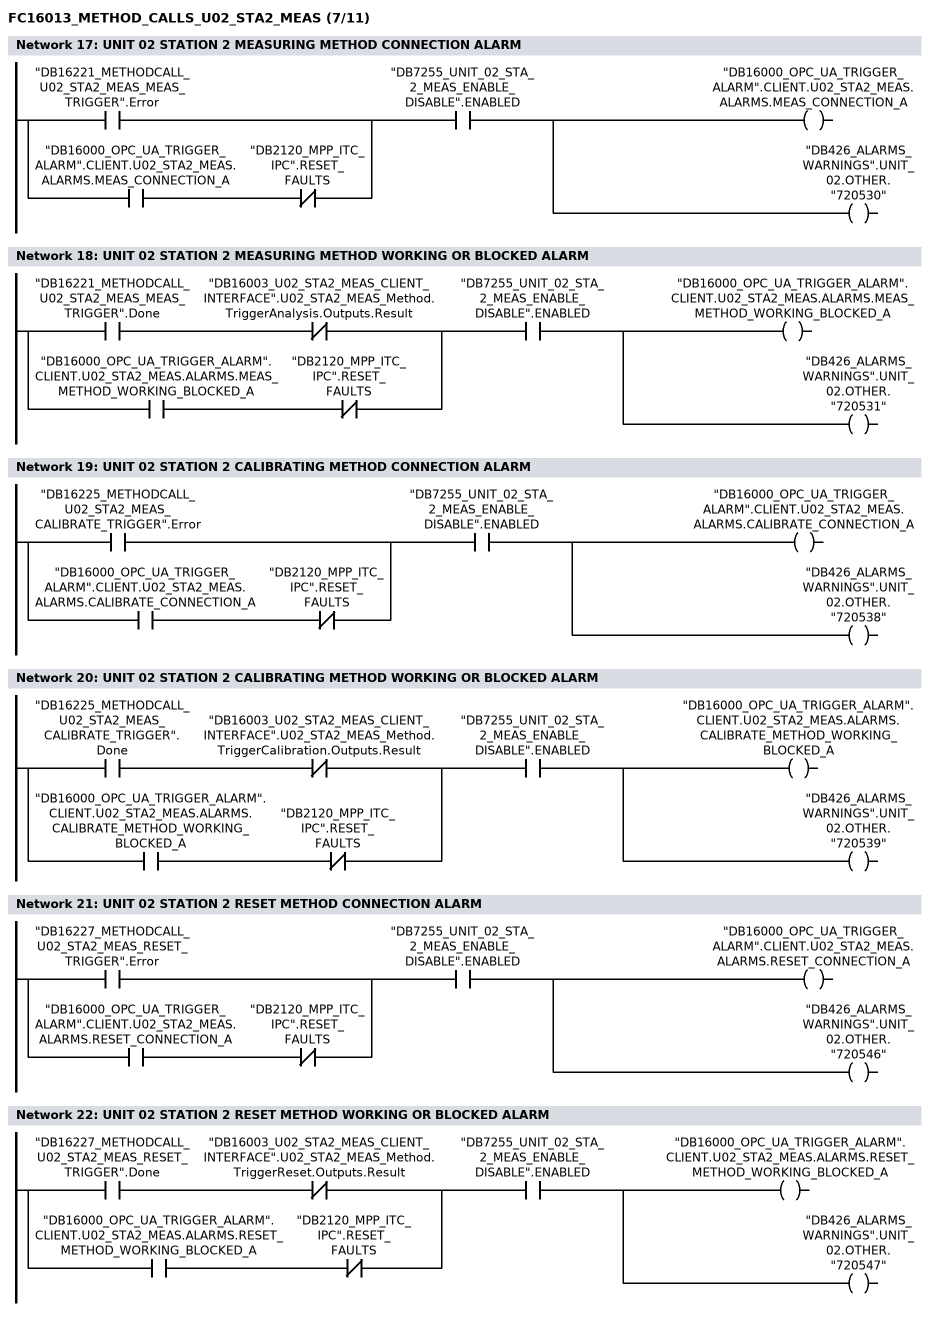
   RUNG wire#powerrail
      Contact( "DB16221_METHODCALL_U02_STA2_MEAS_MEAS_TRIGGER".Error )
      wire#w1
      Contact( "DB7255_UNIT_02_STA_2_MEAS_ENABLE_DISABLE".ENABLED )
      wire#w2
      Coil( "DB16000_OPC_UA_TRIGGER_ALARM".CLIENT.U02_STA2_MEAS.ALARMS.MEAS_CONNECTION_A )
   END_RUNG
   RUNG wire#powerrail
      Contact( "DB16000_OPC_UA_TRIGGER_ALARM".CLIENT.U02_STA2_MEAS.ALARMS.MEAS_CONNECTION_A )
      I_Contact( "DB2120_MPP_ITC_IPC".RESET_FAULTS )
   END_RUNG wire#w1
   RUNG wire#w2
      Coil( "DB426_ALARMS_WARNINGS".UNIT_02.OTHER."720530" )
   END_RUNG
   // the same network as SCL:
   "DB16000_OPC_UA_TRIGGER_ALARM".CLIENT.U02_STA2_MEAS.ALARMS.MEAS_CONNECTION_A := ("DB16221_METHODCALL_U02_STA2_MEAS_MEAS_TRIGGER".Error OR ("DB16000_OPC_UA_TRIGGER_ALARM".CLIENT.U02_STA2_MEAS.ALARMS.MEAS_CONNECTION_A AND NOT "DB2120_MPP_ITC_IPC".RESET_FAULTS)) AND "DB7255_UNIT_02_STA_2_MEAS_ENABLE_DISABLE".ENABLED;
   "DB426_ALARMS_WARNINGS".UNIT_02.OTHER."720530" := "DB16000_OPC_UA_TRIGGER_ALARM".CLIENT.U02_STA2_MEAS.ALARMS.MEAS_CONNECTION_A;
END_REGION

REGION Network 18: UNIT 02 STATION 2 MEASURING METHOD WORKING OR BLOCKED ALARM
   RUNG wire#powerrail
      Contact( "DB16221_METHODCALL_U02_STA2_MEAS_MEAS_TRIGGER".Done )
      I_Contact( "DB16003_U02_STA2_MEAS_CLIENT_INTERFACE".U02_STA2_MEAS_Method.TriggerAnalysis.Outputs.Result )
      wire#w1
      Contact( "DB7255_UNIT_02_STA_2_MEAS_ENABLE_DISABLE".ENABLED )
      wire#w2
      Coil( "DB16000_OPC_UA_TRIGGER_ALARM".CLIENT.U02_STA2_MEAS.ALARMS.MEAS_METHOD_WORKING_BLOCKED_A )
   END_RUNG
   RUNG wire#powerrail
      Contact( "DB16000_OPC_UA_TRIGGER_ALARM".CLIENT.U02_STA2_MEAS.ALARMS.MEAS_METHOD_WORKING_BLOCKED_A )
      I_Contact( "DB2120_MPP_ITC_IPC".RESET_FAULTS )
   END_RUNG wire#w1
   RUNG wire#w2
      Coil( "DB426_ALARMS_WARNINGS".UNIT_02.OTHER."720531" )
   END_RUNG
   // the same network as SCL:
   "DB16000_OPC_UA_TRIGGER_ALARM".CLIENT.U02_STA2_MEAS.ALARMS.MEAS_METHOD_WORKING_BLOCKED_A := (("DB16221_METHODCALL_U02_STA2_MEAS_MEAS_TRIGGER".Done AND NOT "DB16003_U02_STA2_MEAS_CLIENT_INTERFACE".U02_STA2_MEAS_Method.TriggerAnalysis.Outputs.Result) OR ("DB16000_OPC_UA_TRIGGER_ALARM".CLIENT.U02_STA2_MEAS.ALARMS.MEAS_METHOD_WORKING_BLOCKED_A AND NOT "DB2120_MPP_ITC_IPC".RESET_FAULTS)) AND "DB7255_UNIT_02_STA_2_MEAS_ENABLE_DISABLE".ENABLED;
   "DB426_ALARMS_WARNINGS".UNIT_02.OTHER."720531" := "DB16000_OPC_UA_TRIGGER_ALARM".CLIENT.U02_STA2_MEAS.ALARMS.MEAS_METHOD_WORKING_BLOCKED_A;
END_REGION

REGION Network 19: UNIT 02 STATION 2 CALIBRATING METHOD CONNECTION ALARM
   RUNG wire#powerrail
      Contact( "DB16225_METHODCALL_U02_STA2_MEAS_CALIBRATE_TRIGGER".Error )
      wire#w1
      Contact( "DB7255_UNIT_02_STA_2_MEAS_ENABLE_DISABLE".ENABLED )
      wire#w2
      Coil( "DB16000_OPC_UA_TRIGGER_ALARM".CLIENT.U02_STA2_MEAS.ALARMS.CALIBRATE_CONNECTION_A )
   END_RUNG
   RUNG wire#powerrail
      Contact( "DB16000_OPC_UA_TRIGGER_ALARM".CLIENT.U02_STA2_MEAS.ALARMS.CALIBRATE_CONNECTION_A )
      I_Contact( "DB2120_MPP_ITC_IPC".RESET_FAULTS )
   END_RUNG wire#w1
   RUNG wire#w2
      Coil( "DB426_ALARMS_WARNINGS".UNIT_02.OTHER."720538" )
   END_RUNG
   // the same network as SCL:
   "DB16000_OPC_UA_TRIGGER_ALARM".CLIENT.U02_STA2_MEAS.ALARMS.CALIBRATE_CONNECTION_A := ("DB16225_METHODCALL_U02_STA2_MEAS_CALIBRATE_TRIGGER".Error OR ("DB16000_OPC_UA_TRIGGER_ALARM".CLIENT.U02_STA2_MEAS.ALARMS.CALIBRATE_CONNECTION_A AND NOT "DB2120_MPP_ITC_IPC".RESET_FAULTS)) AND "DB7255_UNIT_02_STA_2_MEAS_ENABLE_DISABLE".ENABLED;
   "DB426_ALARMS_WARNINGS".UNIT_02.OTHER."720538" := "DB16000_OPC_UA_TRIGGER_ALARM".CLIENT.U02_STA2_MEAS.ALARMS.CALIBRATE_CONNECTION_A;
END_REGION

REGION Network 20: UNIT 02 STATION 2 CALIBRATING METHOD WORKING OR BLOCKED ALARM
   RUNG wire#powerrail
      Contact( "DB16225_METHODCALL_U02_STA2_MEAS_CALIBRATE_TRIGGER".Done )
      I_Contact( "DB16003_U02_STA2_MEAS_CLIENT_INTERFACE".U02_STA2_MEAS_Method.TriggerCalibration.Outputs.Result )
      wire#w1
      Contact( "DB7255_UNIT_02_STA_2_MEAS_ENABLE_DISABLE".ENABLED )
      wire#w2
      Coil( "DB16000_OPC_UA_TRIGGER_ALARM".CLIENT.U02_STA2_MEAS.ALARMS.CALIBRATE_METHOD_WORKING_BLOCKED_A )
   END_RUNG
   RUNG wire#powerrail
      Contact( "DB16000_OPC_UA_TRIGGER_ALARM".CLIENT.U02_STA2_MEAS.ALARMS.CALIBRATE_METHOD_WORKING_BLOCKED_A )
      I_Contact( "DB2120_MPP_ITC_IPC".RESET_FAULTS )
   END_RUNG wire#w1
   RUNG wire#w2
      Coil( "DB426_ALARMS_WARNINGS".UNIT_02.OTHER."720539" )
   END_RUNG
   // the same network as SCL:
   "DB16000_OPC_UA_TRIGGER_ALARM".CLIENT.U02_STA2_MEAS.ALARMS.CALIBRATE_METHOD_WORKING_BLOCKED_A := (("DB16225_METHODCALL_U02_STA2_MEAS_CALIBRATE_TRIGGER".Done AND NOT "DB16003_U02_STA2_MEAS_CLIENT_INTERFACE".U02_STA2_MEAS_Method.TriggerCalibration.Outputs.Result) OR ("DB16000_OPC_UA_TRIGGER_ALARM".CLIENT.U02_STA2_MEAS.ALARMS.CALIBRATE_METHOD_WORKING_BLOCKED_A AND NOT "DB2120_MPP_ITC_IPC".RESET_FAULTS)) AND "DB7255_UNIT_02_STA_2_MEAS_ENABLE_DISABLE".ENABLED;
   "DB426_ALARMS_WARNINGS".UNIT_02.OTHER."720539" := "DB16000_OPC_UA_TRIGGER_ALARM".CLIENT.U02_STA2_MEAS.ALARMS.CALIBRATE_METHOD_WORKING_BLOCKED_A;
END_REGION

REGION Network 21: UNIT 02 STATION 2 RESET METHOD CONNECTION ALARM
   RUNG wire#powerrail
      Contact( "DB16227_METHODCALL_U02_STA2_MEAS_RESET_TRIGGER".Error )
      wire#w1
      Contact( "DB7255_UNIT_02_STA_2_MEAS_ENABLE_DISABLE".ENABLED )
      wire#w2
      Coil( "DB16000_OPC_UA_TRIGGER_ALARM".CLIENT.U02_STA2_MEAS.ALARMS.RESET_CONNECTION_A )
   END_RUNG
   RUNG wire#powerrail
      Contact( "DB16000_OPC_UA_TRIGGER_ALARM".CLIENT.U02_STA2_MEAS.ALARMS.RESET_CONNECTION_A )
      I_Contact( "DB2120_MPP_ITC_IPC".RESET_FAULTS )
   END_RUNG wire#w1
   RUNG wire#w2
      Coil( "DB426_ALARMS_WARNINGS".UNIT_02.OTHER."720546" )
   END_RUNG
   // the same network as SCL:
   "DB16000_OPC_UA_TRIGGER_ALARM".CLIENT.U02_STA2_MEAS.ALARMS.RESET_CONNECTION_A := ("DB16227_METHODCALL_U02_STA2_MEAS_RESET_TRIGGER".Error OR ("DB16000_OPC_UA_TRIGGER_ALARM".CLIENT.U02_STA2_MEAS.ALARMS.RESET_CONNECTION_A AND NOT "DB2120_MPP_ITC_IPC".RESET_FAULTS)) AND "DB7255_UNIT_02_STA_2_MEAS_ENABLE_DISABLE".ENABLED;
   "DB426_ALARMS_WARNINGS".UNIT_02.OTHER."720546" := "DB16000_OPC_UA_TRIGGER_ALARM".CLIENT.U02_STA2_MEAS.ALARMS.RESET_CONNECTION_A;
END_REGION

REGION Network 22: UNIT 02 STATION 2 RESET METHOD WORKING OR BLOCKED ALARM
   RUNG wire#powerrail
      Contact( "DB16227_METHODCALL_U02_STA2_MEAS_RESET_TRIGGER".Done )
      I_Contact( "DB16003_U02_STA2_MEAS_CLIENT_INTERFACE".U02_STA2_MEAS_Method.TriggerReset.Outputs.Result )
      wire#w1
      Contact( "DB7255_UNIT_02_STA_2_MEAS_ENABLE_DISABLE".ENABLED )
      wire#w2
      Coil( "DB16000_OPC_UA_TRIGGER_ALARM".CLIENT.U02_STA2_MEAS.ALARMS.RESET_METHOD_WORKING_BLOCKED_A )
   END_RUNG
   RUNG wire#powerrail
      Contact( "DB16000_OPC_UA_TRIGGER_ALARM".CLIENT.U02_STA2_MEAS.ALARMS.RESET_METHOD_WORKING_BLOCKED_A )
      I_Contact( "DB2120_MPP_ITC_IPC".RESET_FAULTS )
   END_RUNG wire#w1
   RUNG wire#w2
      Coil( "DB426_ALARMS_WARNINGS".UNIT_02.OTHER."720547" )
   END_RUNG
   // the same network as SCL:
   "DB16000_OPC_UA_TRIGGER_ALARM".CLIENT.U02_STA2_MEAS.ALARMS.RESET_METHOD_WORKING_BLOCKED_A := (("DB16227_METHODCALL_U02_STA2_MEAS_RESET_TRIGGER".Done AND NOT "DB16003_U02_STA2_MEAS_CLIENT_INTERFACE".U02_STA2_MEAS_Method.TriggerReset.Outputs.Result) OR ("DB16000_OPC_UA_TRIGGER_ALARM".CLIENT.U02_STA2_MEAS.ALARMS.RESET_METHOD_WORKING_BLOCKED_A AND NOT "DB2120_MPP_ITC_IPC".RESET_FAULTS)) AND "DB7255_UNIT_02_STA_2_MEAS_ENABLE_DISABLE".ENABLED;
   "DB426_ALARMS_WARNINGS".UNIT_02.OTHER."720547" := "DB16000_OPC_UA_TRIGGER_ALARM".CLIENT.U02_STA2_MEAS.ALARMS.RESET_METHOD_WORKING_BLOCKED_A;
END_REGION

REGION Network 23: UNIT 02 STATION 2 READ VARIABLES CONNECTION ALARM
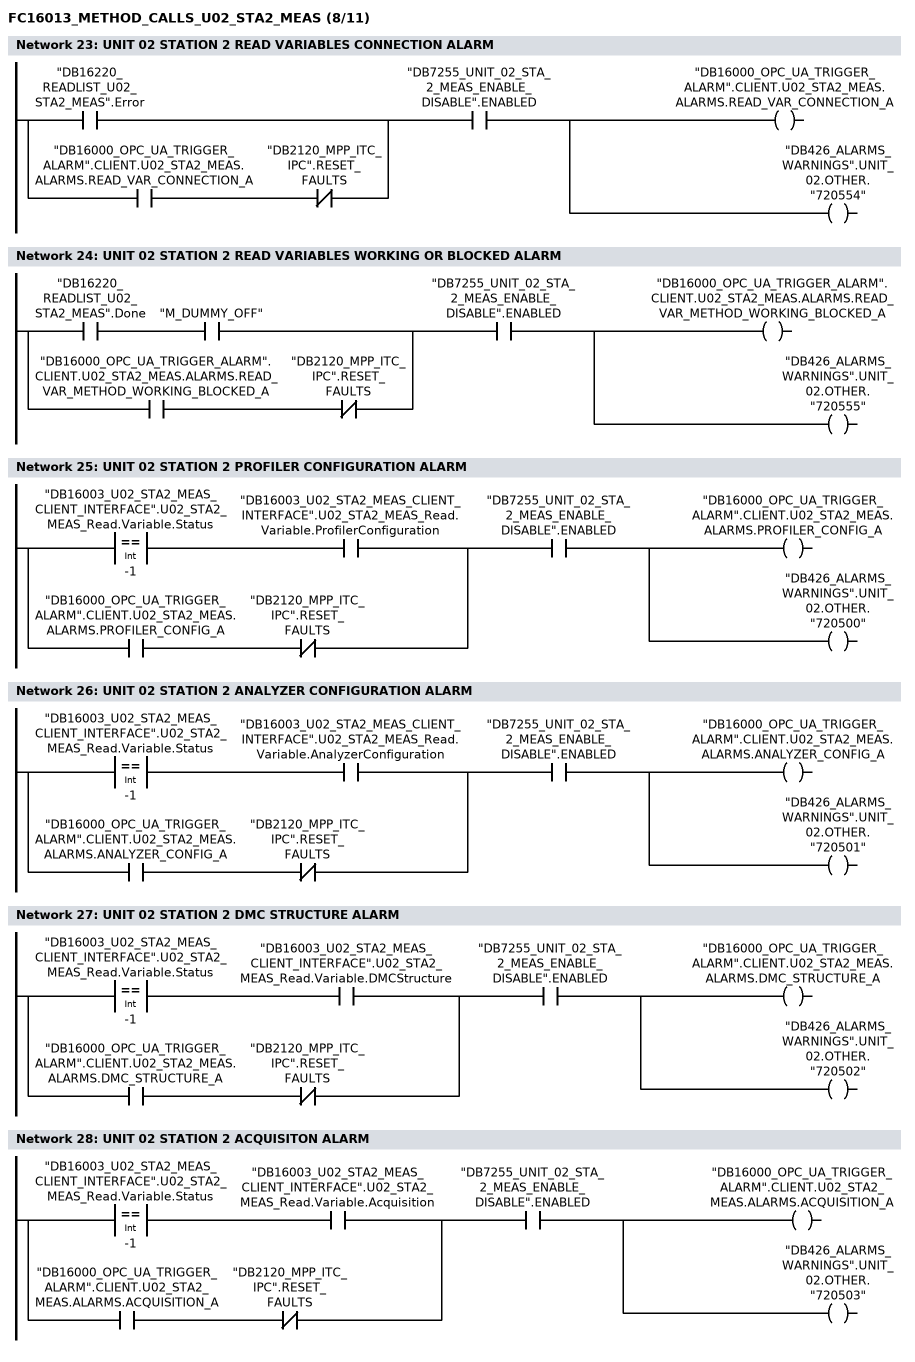
   RUNG wire#powerrail
      Contact( "DB16220_READLIST_U02_STA2_MEAS".Error )
      wire#w1
      Contact( "DB7255_UNIT_02_STA_2_MEAS_ENABLE_DISABLE".ENABLED )
      wire#w2
      Coil( "DB16000_OPC_UA_TRIGGER_ALARM".CLIENT.U02_STA2_MEAS.ALARMS.READ_VAR_CONNECTION_A )
   END_RUNG
   RUNG wire#powerrail
      Contact( "DB16000_OPC_UA_TRIGGER_ALARM".CLIENT.U02_STA2_MEAS.ALARMS.READ_VAR_CONNECTION_A )
      I_Contact( "DB2120_MPP_ITC_IPC".RESET_FAULTS )
   END_RUNG wire#w1
   RUNG wire#w2
      Coil( "DB426_ALARMS_WARNINGS".UNIT_02.OTHER."720554" )
   END_RUNG
   // the same network as SCL:
   "DB16000_OPC_UA_TRIGGER_ALARM".CLIENT.U02_STA2_MEAS.ALARMS.READ_VAR_CONNECTION_A := ("DB16220_READLIST_U02_STA2_MEAS".Error OR ("DB16000_OPC_UA_TRIGGER_ALARM".CLIENT.U02_STA2_MEAS.ALARMS.READ_VAR_CONNECTION_A AND NOT "DB2120_MPP_ITC_IPC".RESET_FAULTS)) AND "DB7255_UNIT_02_STA_2_MEAS_ENABLE_DISABLE".ENABLED;
   "DB426_ALARMS_WARNINGS".UNIT_02.OTHER."720554" := "DB16000_OPC_UA_TRIGGER_ALARM".CLIENT.U02_STA2_MEAS.ALARMS.READ_VAR_CONNECTION_A;
END_REGION

REGION Network 24: UNIT 02 STATION 2 READ VARIABLES WORKING OR BLOCKED ALARM
   RUNG wire#powerrail
      Contact( "DB16220_READLIST_U02_STA2_MEAS".Done )
      Contact( "M_DUMMY_OFF" )
      wire#w1
      Contact( "DB7255_UNIT_02_STA_2_MEAS_ENABLE_DISABLE".ENABLED )
      wire#w2
      Coil( "DB16000_OPC_UA_TRIGGER_ALARM".CLIENT.U02_STA2_MEAS.ALARMS.READ_VAR_METHOD_WORKING_BLOCKED_A )
   END_RUNG
   RUNG wire#powerrail
      Contact( "DB16000_OPC_UA_TRIGGER_ALARM".CLIENT.U02_STA2_MEAS.ALARMS.READ_VAR_METHOD_WORKING_BLOCKED_A )
      I_Contact( "DB2120_MPP_ITC_IPC".RESET_FAULTS )
   END_RUNG wire#w1
   RUNG wire#w2
      Coil( "DB426_ALARMS_WARNINGS".UNIT_02.OTHER."720555" )
   END_RUNG
   // the same network as SCL:
   "DB16000_OPC_UA_TRIGGER_ALARM".CLIENT.U02_STA2_MEAS.ALARMS.READ_VAR_METHOD_WORKING_BLOCKED_A := (("DB16220_READLIST_U02_STA2_MEAS".Done AND "M_DUMMY_OFF") OR ("DB16000_OPC_UA_TRIGGER_ALARM".CLIENT.U02_STA2_MEAS.ALARMS.READ_VAR_METHOD_WORKING_BLOCKED_A AND NOT "DB2120_MPP_ITC_IPC".RESET_FAULTS)) AND "DB7255_UNIT_02_STA_2_MEAS_ENABLE_DISABLE".ENABLED;
   "DB426_ALARMS_WARNINGS".UNIT_02.OTHER."720555" := "DB16000_OPC_UA_TRIGGER_ALARM".CLIENT.U02_STA2_MEAS.ALARMS.READ_VAR_METHOD_WORKING_BLOCKED_A;
END_REGION

REGION Network 25: UNIT 02 STATION 2 PROFILER CONFIGURATION ALARM
   RUNG wire#powerrail
      { S7_Templates := "SrcType := Int" } EQ_Contact(in1 := "DB16003_U02_STA2_MEAS_CLIENT_INTERFACE".U02_STA2_MEAS_Read.Variable.Status, in2 := -1)
      Contact( "DB16003_U02_STA2_MEAS_CLIENT_INTERFACE".U02_STA2_MEAS_Read.Variable.ProfilerConfiguration )
      wire#w1
      Contact( "DB7255_UNIT_02_STA_2_MEAS_ENABLE_DISABLE".ENABLED )
      wire#w2
      Coil( "DB16000_OPC_UA_TRIGGER_ALARM".CLIENT.U02_STA2_MEAS.ALARMS.PROFILER_CONFIG_A )
   END_RUNG
   RUNG wire#powerrail
      Contact( "DB16000_OPC_UA_TRIGGER_ALARM".CLIENT.U02_STA2_MEAS.ALARMS.PROFILER_CONFIG_A )
      I_Contact( "DB2120_MPP_ITC_IPC".RESET_FAULTS )
   END_RUNG wire#w1
   RUNG wire#w2
      Coil( "DB426_ALARMS_WARNINGS".UNIT_02.OTHER."720500" )
   END_RUNG
   // the same network as SCL:
   "DB16000_OPC_UA_TRIGGER_ALARM".CLIENT.U02_STA2_MEAS.ALARMS.PROFILER_CONFIG_A := ((("DB16003_U02_STA2_MEAS_CLIENT_INTERFACE".U02_STA2_MEAS_Read.Variable.Status = (-1)) AND "DB16003_U02_STA2_MEAS_CLIENT_INTERFACE".U02_STA2_MEAS_Read.Variable.ProfilerConfiguration) OR ("DB16000_OPC_UA_TRIGGER_ALARM".CLIENT.U02_STA2_MEAS.ALARMS.PROFILER_CONFIG_A AND NOT "DB2120_MPP_ITC_IPC".RESET_FAULTS)) AND "DB7255_UNIT_02_STA_2_MEAS_ENABLE_DISABLE".ENABLED;
   "DB426_ALARMS_WARNINGS".UNIT_02.OTHER."720500" := "DB16000_OPC_UA_TRIGGER_ALARM".CLIENT.U02_STA2_MEAS.ALARMS.PROFILER_CONFIG_A;
END_REGION

REGION Network 26: UNIT 02 STATION 2 ANALYZER CONFIGURATION ALARM
   RUNG wire#powerrail
      { S7_Templates := "SrcType := Int" } EQ_Contact(in1 := "DB16003_U02_STA2_MEAS_CLIENT_INTERFACE".U02_STA2_MEAS_Read.Variable.Status, in2 := -1)
      Contact( "DB16003_U02_STA2_MEAS_CLIENT_INTERFACE".U02_STA2_MEAS_Read.Variable.AnalyzerConfiguration )
      wire#w1
      Contact( "DB7255_UNIT_02_STA_2_MEAS_ENABLE_DISABLE".ENABLED )
      wire#w2
      Coil( "DB16000_OPC_UA_TRIGGER_ALARM".CLIENT.U02_STA2_MEAS.ALARMS.ANALYZER_CONFIG_A )
   END_RUNG
   RUNG wire#powerrail
      Contact( "DB16000_OPC_UA_TRIGGER_ALARM".CLIENT.U02_STA2_MEAS.ALARMS.ANALYZER_CONFIG_A )
      I_Contact( "DB2120_MPP_ITC_IPC".RESET_FAULTS )
   END_RUNG wire#w1
   RUNG wire#w2
      Coil( "DB426_ALARMS_WARNINGS".UNIT_02.OTHER."720501" )
   END_RUNG
   // the same network as SCL:
   "DB16000_OPC_UA_TRIGGER_ALARM".CLIENT.U02_STA2_MEAS.ALARMS.ANALYZER_CONFIG_A := ((("DB16003_U02_STA2_MEAS_CLIENT_INTERFACE".U02_STA2_MEAS_Read.Variable.Status = (-1)) AND "DB16003_U02_STA2_MEAS_CLIENT_INTERFACE".U02_STA2_MEAS_Read.Variable.AnalyzerConfiguration) OR ("DB16000_OPC_UA_TRIGGER_ALARM".CLIENT.U02_STA2_MEAS.ALARMS.ANALYZER_CONFIG_A AND NOT "DB2120_MPP_ITC_IPC".RESET_FAULTS)) AND "DB7255_UNIT_02_STA_2_MEAS_ENABLE_DISABLE".ENABLED;
   "DB426_ALARMS_WARNINGS".UNIT_02.OTHER."720501" := "DB16000_OPC_UA_TRIGGER_ALARM".CLIENT.U02_STA2_MEAS.ALARMS.ANALYZER_CONFIG_A;
END_REGION

REGION Network 27: UNIT 02 STATION 2 DMC STRUCTURE ALARM
   RUNG wire#powerrail
      { S7_Templates := "SrcType := Int" } EQ_Contact(in1 := "DB16003_U02_STA2_MEAS_CLIENT_INTERFACE".U02_STA2_MEAS_Read.Variable.Status, in2 := -1)
      Contact( "DB16003_U02_STA2_MEAS_CLIENT_INTERFACE".U02_STA2_MEAS_Read.Variable.DMCStructure )
      wire#w1
      Contact( "DB7255_UNIT_02_STA_2_MEAS_ENABLE_DISABLE".ENABLED )
      wire#w2
      Coil( "DB16000_OPC_UA_TRIGGER_ALARM".CLIENT.U02_STA2_MEAS.ALARMS.DMC_STRUCTURE_A )
   END_RUNG
   RUNG wire#powerrail
      Contact( "DB16000_OPC_UA_TRIGGER_ALARM".CLIENT.U02_STA2_MEAS.ALARMS.DMC_STRUCTURE_A )
      I_Contact( "DB2120_MPP_ITC_IPC".RESET_FAULTS )
   END_RUNG wire#w1
   RUNG wire#w2
      Coil( "DB426_ALARMS_WARNINGS".UNIT_02.OTHER."720502" )
   END_RUNG
   // the same network as SCL:
   "DB16000_OPC_UA_TRIGGER_ALARM".CLIENT.U02_STA2_MEAS.ALARMS.DMC_STRUCTURE_A := ((("DB16003_U02_STA2_MEAS_CLIENT_INTERFACE".U02_STA2_MEAS_Read.Variable.Status = (-1)) AND "DB16003_U02_STA2_MEAS_CLIENT_INTERFACE".U02_STA2_MEAS_Read.Variable.DMCStructure) OR ("DB16000_OPC_UA_TRIGGER_ALARM".CLIENT.U02_STA2_MEAS.ALARMS.DMC_STRUCTURE_A AND NOT "DB2120_MPP_ITC_IPC".RESET_FAULTS)) AND "DB7255_UNIT_02_STA_2_MEAS_ENABLE_DISABLE".ENABLED;
   "DB426_ALARMS_WARNINGS".UNIT_02.OTHER."720502" := "DB16000_OPC_UA_TRIGGER_ALARM".CLIENT.U02_STA2_MEAS.ALARMS.DMC_STRUCTURE_A;
END_REGION

REGION Network 28: UNIT 02 STATION 2 ACQUISITON ALARM
   RUNG wire#powerrail
      { S7_Templates := "SrcType := Int" } EQ_Contact(in1 := "DB16003_U02_STA2_MEAS_CLIENT_INTERFACE".U02_STA2_MEAS_Read.Variable.Status, in2 := -1)
      Contact( "DB16003_U02_STA2_MEAS_CLIENT_INTERFACE".U02_STA2_MEAS_Read.Variable.Acquisition )
      wire#w1
      Contact( "DB7255_UNIT_02_STA_2_MEAS_ENABLE_DISABLE".ENABLED )
      wire#w2
      Coil( "DB16000_OPC_UA_TRIGGER_ALARM".CLIENT.U02_STA2_MEAS.ALARMS.ACQUISITION_A )
   END_RUNG
   RUNG wire#powerrail
      Contact( "DB16000_OPC_UA_TRIGGER_ALARM".CLIENT.U02_STA2_MEAS.ALARMS.ACQUISITION_A )
      I_Contact( "DB2120_MPP_ITC_IPC".RESET_FAULTS )
   END_RUNG wire#w1
   RUNG wire#w2
      Coil( "DB426_ALARMS_WARNINGS".UNIT_02.OTHER."720503" )
   END_RUNG
   // the same network as SCL:
   "DB16000_OPC_UA_TRIGGER_ALARM".CLIENT.U02_STA2_MEAS.ALARMS.ACQUISITION_A := ((("DB16003_U02_STA2_MEAS_CLIENT_INTERFACE".U02_STA2_MEAS_Read.Variable.Status = (-1)) AND "DB16003_U02_STA2_MEAS_CLIENT_INTERFACE".U02_STA2_MEAS_Read.Variable.Acquisition) OR ("DB16000_OPC_UA_TRIGGER_ALARM".CLIENT.U02_STA2_MEAS.ALARMS.ACQUISITION_A AND NOT "DB2120_MPP_ITC_IPC".RESET_FAULTS)) AND "DB7255_UNIT_02_STA_2_MEAS_ENABLE_DISABLE".ENABLED;
   "DB426_ALARMS_WARNINGS".UNIT_02.OTHER."720503" := "DB16000_OPC_UA_TRIGGER_ALARM".CLIENT.U02_STA2_MEAS.ALARMS.ACQUISITION_A;
END_REGION

REGION Network 29: UNIT 02 STATION 2 PROFILER INITIALIZTION ALARM
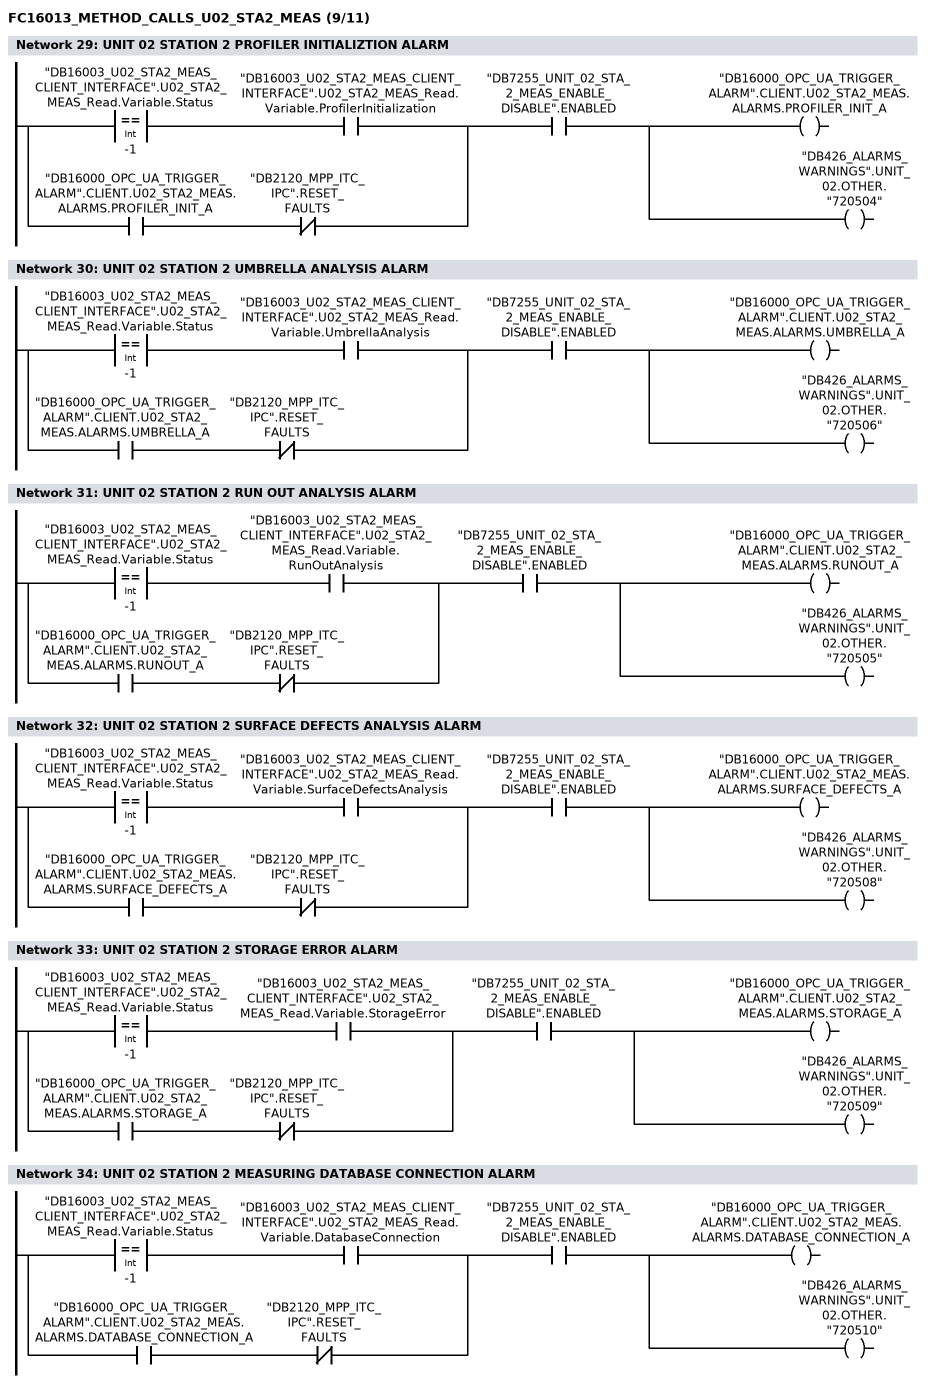
   RUNG wire#powerrail
      { S7_Templates := "SrcType := Int" } EQ_Contact(in1 := "DB16003_U02_STA2_MEAS_CLIENT_INTERFACE".U02_STA2_MEAS_Read.Variable.Status, in2 := -1)
      Contact( "DB16003_U02_STA2_MEAS_CLIENT_INTERFACE".U02_STA2_MEAS_Read.Variable.ProfilerInitialization )
      wire#w1
      Contact( "DB7255_UNIT_02_STA_2_MEAS_ENABLE_DISABLE".ENABLED )
      wire#w2
      Coil( "DB16000_OPC_UA_TRIGGER_ALARM".CLIENT.U02_STA2_MEAS.ALARMS.PROFILER_INIT_A )
   END_RUNG
   RUNG wire#powerrail
      Contact( "DB16000_OPC_UA_TRIGGER_ALARM".CLIENT.U02_STA2_MEAS.ALARMS.PROFILER_INIT_A )
      I_Contact( "DB2120_MPP_ITC_IPC".RESET_FAULTS )
   END_RUNG wire#w1
   RUNG wire#w2
      Coil( "DB426_ALARMS_WARNINGS".UNIT_02.OTHER."720504" )
   END_RUNG
   // the same network as SCL:
   "DB16000_OPC_UA_TRIGGER_ALARM".CLIENT.U02_STA2_MEAS.ALARMS.PROFILER_INIT_A := ((("DB16003_U02_STA2_MEAS_CLIENT_INTERFACE".U02_STA2_MEAS_Read.Variable.Status = (-1)) AND "DB16003_U02_STA2_MEAS_CLIENT_INTERFACE".U02_STA2_MEAS_Read.Variable.ProfilerInitialization) OR ("DB16000_OPC_UA_TRIGGER_ALARM".CLIENT.U02_STA2_MEAS.ALARMS.PROFILER_INIT_A AND NOT "DB2120_MPP_ITC_IPC".RESET_FAULTS)) AND "DB7255_UNIT_02_STA_2_MEAS_ENABLE_DISABLE".ENABLED;
   "DB426_ALARMS_WARNINGS".UNIT_02.OTHER."720504" := "DB16000_OPC_UA_TRIGGER_ALARM".CLIENT.U02_STA2_MEAS.ALARMS.PROFILER_INIT_A;
END_REGION

REGION Network 30: UNIT 02 STATION 2 UMBRELLA ANALYSIS ALARM
   RUNG wire#powerrail
      { S7_Templates := "SrcType := Int" } EQ_Contact(in1 := "DB16003_U02_STA2_MEAS_CLIENT_INTERFACE".U02_STA2_MEAS_Read.Variable.Status, in2 := -1)
      Contact( "DB16003_U02_STA2_MEAS_CLIENT_INTERFACE".U02_STA2_MEAS_Read.Variable.UmbrellaAnalysis )
      wire#w1
      Contact( "DB7255_UNIT_02_STA_2_MEAS_ENABLE_DISABLE".ENABLED )
      wire#w2
      Coil( "DB16000_OPC_UA_TRIGGER_ALARM".CLIENT.U02_STA2_MEAS.ALARMS.UMBRELLA_A )
   END_RUNG
   RUNG wire#powerrail
      Contact( "DB16000_OPC_UA_TRIGGER_ALARM".CLIENT.U02_STA2_MEAS.ALARMS.UMBRELLA_A )
      I_Contact( "DB2120_MPP_ITC_IPC".RESET_FAULTS )
   END_RUNG wire#w1
   RUNG wire#w2
      Coil( "DB426_ALARMS_WARNINGS".UNIT_02.OTHER."720506" )
   END_RUNG
   // the same network as SCL:
   "DB16000_OPC_UA_TRIGGER_ALARM".CLIENT.U02_STA2_MEAS.ALARMS.UMBRELLA_A := ((("DB16003_U02_STA2_MEAS_CLIENT_INTERFACE".U02_STA2_MEAS_Read.Variable.Status = (-1)) AND "DB16003_U02_STA2_MEAS_CLIENT_INTERFACE".U02_STA2_MEAS_Read.Variable.UmbrellaAnalysis) OR ("DB16000_OPC_UA_TRIGGER_ALARM".CLIENT.U02_STA2_MEAS.ALARMS.UMBRELLA_A AND NOT "DB2120_MPP_ITC_IPC".RESET_FAULTS)) AND "DB7255_UNIT_02_STA_2_MEAS_ENABLE_DISABLE".ENABLED;
   "DB426_ALARMS_WARNINGS".UNIT_02.OTHER."720506" := "DB16000_OPC_UA_TRIGGER_ALARM".CLIENT.U02_STA2_MEAS.ALARMS.UMBRELLA_A;
END_REGION

REGION Network 31: UNIT 02 STATION 2 RUN OUT ANALYSIS ALARM
   RUNG wire#powerrail
      { S7_Templates := "SrcType := Int" } EQ_Contact(in1 := "DB16003_U02_STA2_MEAS_CLIENT_INTERFACE".U02_STA2_MEAS_Read.Variable.Status, in2 := -1)
      Contact( "DB16003_U02_STA2_MEAS_CLIENT_INTERFACE".U02_STA2_MEAS_Read.Variable.RunOutAnalysis )
      wire#w1
      Contact( "DB7255_UNIT_02_STA_2_MEAS_ENABLE_DISABLE".ENABLED )
      wire#w2
      Coil( "DB16000_OPC_UA_TRIGGER_ALARM".CLIENT.U02_STA2_MEAS.ALARMS.RUNOUT_A )
   END_RUNG
   RUNG wire#powerrail
      Contact( "DB16000_OPC_UA_TRIGGER_ALARM".CLIENT.U02_STA2_MEAS.ALARMS.RUNOUT_A )
      I_Contact( "DB2120_MPP_ITC_IPC".RESET_FAULTS )
   END_RUNG wire#w1
   RUNG wire#w2
      Coil( "DB426_ALARMS_WARNINGS".UNIT_02.OTHER."720505" )
   END_RUNG
   // the same network as SCL:
   "DB16000_OPC_UA_TRIGGER_ALARM".CLIENT.U02_STA2_MEAS.ALARMS.RUNOUT_A := ((("DB16003_U02_STA2_MEAS_CLIENT_INTERFACE".U02_STA2_MEAS_Read.Variable.Status = (-1)) AND "DB16003_U02_STA2_MEAS_CLIENT_INTERFACE".U02_STA2_MEAS_Read.Variable.RunOutAnalysis) OR ("DB16000_OPC_UA_TRIGGER_ALARM".CLIENT.U02_STA2_MEAS.ALARMS.RUNOUT_A AND NOT "DB2120_MPP_ITC_IPC".RESET_FAULTS)) AND "DB7255_UNIT_02_STA_2_MEAS_ENABLE_DISABLE".ENABLED;
   "DB426_ALARMS_WARNINGS".UNIT_02.OTHER."720505" := "DB16000_OPC_UA_TRIGGER_ALARM".CLIENT.U02_STA2_MEAS.ALARMS.RUNOUT_A;
END_REGION

REGION Network 32: UNIT 02 STATION 2 SURFACE DEFECTS ANALYSIS ALARM
   RUNG wire#powerrail
      { S7_Templates := "SrcType := Int" } EQ_Contact(in1 := "DB16003_U02_STA2_MEAS_CLIENT_INTERFACE".U02_STA2_MEAS_Read.Variable.Status, in2 := -1)
      Contact( "DB16003_U02_STA2_MEAS_CLIENT_INTERFACE".U02_STA2_MEAS_Read.Variable.SurfaceDefectsAnalysis )
      wire#w1
      Contact( "DB7255_UNIT_02_STA_2_MEAS_ENABLE_DISABLE".ENABLED )
      wire#w2
      Coil( "DB16000_OPC_UA_TRIGGER_ALARM".CLIENT.U02_STA2_MEAS.ALARMS.SURFACE_DEFECTS_A )
   END_RUNG
   RUNG wire#powerrail
      Contact( "DB16000_OPC_UA_TRIGGER_ALARM".CLIENT.U02_STA2_MEAS.ALARMS.SURFACE_DEFECTS_A )
      I_Contact( "DB2120_MPP_ITC_IPC".RESET_FAULTS )
   END_RUNG wire#w1
   RUNG wire#w2
      Coil( "DB426_ALARMS_WARNINGS".UNIT_02.OTHER."720508" )
   END_RUNG
   // the same network as SCL:
   "DB16000_OPC_UA_TRIGGER_ALARM".CLIENT.U02_STA2_MEAS.ALARMS.SURFACE_DEFECTS_A := ((("DB16003_U02_STA2_MEAS_CLIENT_INTERFACE".U02_STA2_MEAS_Read.Variable.Status = (-1)) AND "DB16003_U02_STA2_MEAS_CLIENT_INTERFACE".U02_STA2_MEAS_Read.Variable.SurfaceDefectsAnalysis) OR ("DB16000_OPC_UA_TRIGGER_ALARM".CLIENT.U02_STA2_MEAS.ALARMS.SURFACE_DEFECTS_A AND NOT "DB2120_MPP_ITC_IPC".RESET_FAULTS)) AND "DB7255_UNIT_02_STA_2_MEAS_ENABLE_DISABLE".ENABLED;
   "DB426_ALARMS_WARNINGS".UNIT_02.OTHER."720508" := "DB16000_OPC_UA_TRIGGER_ALARM".CLIENT.U02_STA2_MEAS.ALARMS.SURFACE_DEFECTS_A;
END_REGION

REGION Network 33: UNIT 02 STATION 2 STORAGE ERROR ALARM
   RUNG wire#powerrail
      { S7_Templates := "SrcType := Int" } EQ_Contact(in1 := "DB16003_U02_STA2_MEAS_CLIENT_INTERFACE".U02_STA2_MEAS_Read.Variable.Status, in2 := -1)
      Contact( "DB16003_U02_STA2_MEAS_CLIENT_INTERFACE".U02_STA2_MEAS_Read.Variable.StorageError )
      wire#w1
      Contact( "DB7255_UNIT_02_STA_2_MEAS_ENABLE_DISABLE".ENABLED )
      wire#w2
      Coil( "DB16000_OPC_UA_TRIGGER_ALARM".CLIENT.U02_STA2_MEAS.ALARMS.STORAGE_A )
   END_RUNG
   RUNG wire#powerrail
      Contact( "DB16000_OPC_UA_TRIGGER_ALARM".CLIENT.U02_STA2_MEAS.ALARMS.STORAGE_A )
      I_Contact( "DB2120_MPP_ITC_IPC".RESET_FAULTS )
   END_RUNG wire#w1
   RUNG wire#w2
      Coil( "DB426_ALARMS_WARNINGS".UNIT_02.OTHER."720509" )
   END_RUNG
   // the same network as SCL:
   "DB16000_OPC_UA_TRIGGER_ALARM".CLIENT.U02_STA2_MEAS.ALARMS.STORAGE_A := ((("DB16003_U02_STA2_MEAS_CLIENT_INTERFACE".U02_STA2_MEAS_Read.Variable.Status = (-1)) AND "DB16003_U02_STA2_MEAS_CLIENT_INTERFACE".U02_STA2_MEAS_Read.Variable.StorageError) OR ("DB16000_OPC_UA_TRIGGER_ALARM".CLIENT.U02_STA2_MEAS.ALARMS.STORAGE_A AND NOT "DB2120_MPP_ITC_IPC".RESET_FAULTS)) AND "DB7255_UNIT_02_STA_2_MEAS_ENABLE_DISABLE".ENABLED;
   "DB426_ALARMS_WARNINGS".UNIT_02.OTHER."720509" := "DB16000_OPC_UA_TRIGGER_ALARM".CLIENT.U02_STA2_MEAS.ALARMS.STORAGE_A;
END_REGION

REGION Network 34: UNIT 02 STATION 2 MEASURING DATABASE CONNECTION ALARM
   RUNG wire#powerrail
      { S7_Templates := "SrcType := Int" } EQ_Contact(in1 := "DB16003_U02_STA2_MEAS_CLIENT_INTERFACE".U02_STA2_MEAS_Read.Variable.Status, in2 := -1)
      Contact( "DB16003_U02_STA2_MEAS_CLIENT_INTERFACE".U02_STA2_MEAS_Read.Variable.DatabaseConnection )
      wire#w1
      Contact( "DB7255_UNIT_02_STA_2_MEAS_ENABLE_DISABLE".ENABLED )
      wire#w2
      Coil( "DB16000_OPC_UA_TRIGGER_ALARM".CLIENT.U02_STA2_MEAS.ALARMS.DATABASE_CONNECTION_A )
   END_RUNG
   RUNG wire#powerrail
      Contact( "DB16000_OPC_UA_TRIGGER_ALARM".CLIENT.U02_STA2_MEAS.ALARMS.DATABASE_CONNECTION_A )
      I_Contact( "DB2120_MPP_ITC_IPC".RESET_FAULTS )
   END_RUNG wire#w1
   RUNG wire#w2
      Coil( "DB426_ALARMS_WARNINGS".UNIT_02.OTHER."720510" )
   END_RUNG
   // the same network as SCL:
   "DB16000_OPC_UA_TRIGGER_ALARM".CLIENT.U02_STA2_MEAS.ALARMS.DATABASE_CONNECTION_A := ((("DB16003_U02_STA2_MEAS_CLIENT_INTERFACE".U02_STA2_MEAS_Read.Variable.Status = (-1)) AND "DB16003_U02_STA2_MEAS_CLIENT_INTERFACE".U02_STA2_MEAS_Read.Variable.DatabaseConnection) OR ("DB16000_OPC_UA_TRIGGER_ALARM".CLIENT.U02_STA2_MEAS.ALARMS.DATABASE_CONNECTION_A AND NOT "DB2120_MPP_ITC_IPC".RESET_FAULTS)) AND "DB7255_UNIT_02_STA_2_MEAS_ENABLE_DISABLE".ENABLED;
   "DB426_ALARMS_WARNINGS".UNIT_02.OTHER."720510" := "DB16000_OPC_UA_TRIGGER_ALARM".CLIENT.U02_STA2_MEAS.ALARMS.DATABASE_CONNECTION_A;
END_REGION

REGION Network 35: UNIT 02 STATION 2 MISSING CALIBRATION IN FIXTURE 1 ALARM
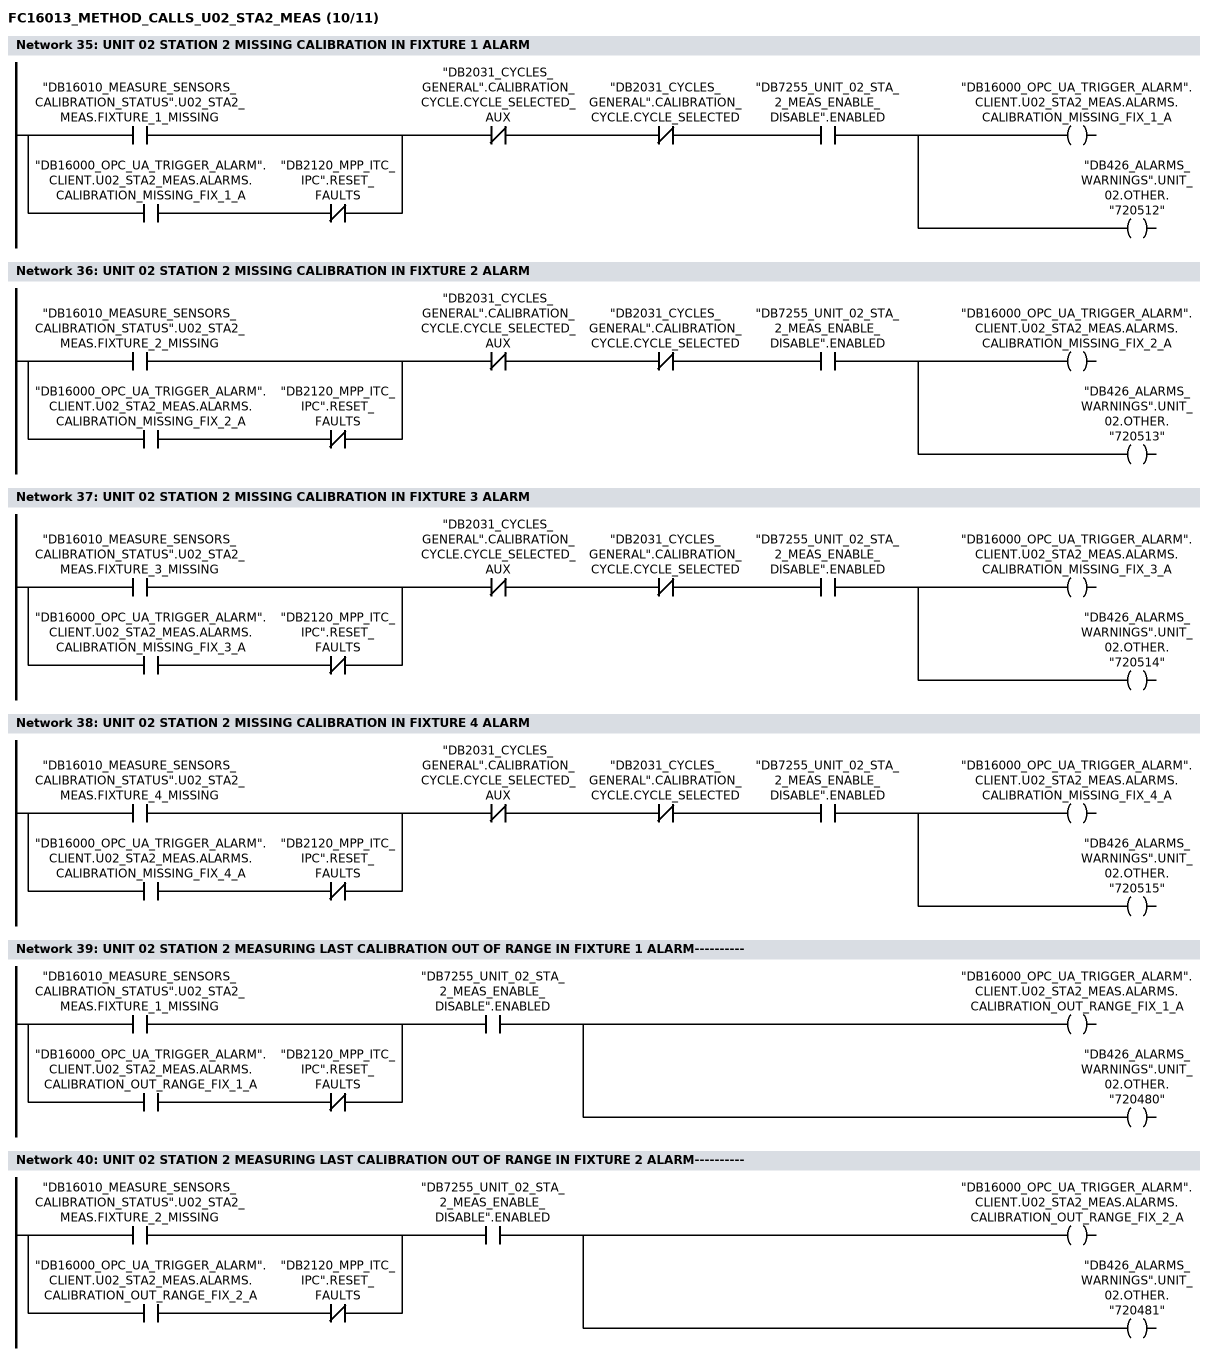
   RUNG wire#powerrail
      Contact( "DB16010_MEASURE_SENSORS_CALIBRATION_STATUS".U02_STA2_MEAS.FIXTURE_1_MISSING )
      wire#w1
      I_Contact( "DB2031_CYCLES_GENERAL".CALIBRATION_CYCLE.CYCLE_SELECTED_AUX )
      I_Contact( "DB2031_CYCLES_GENERAL".CALIBRATION_CYCLE.CYCLE_SELECTED )
      Contact( "DB7255_UNIT_02_STA_2_MEAS_ENABLE_DISABLE".ENABLED )
      wire#w2
      Coil( "DB16000_OPC_UA_TRIGGER_ALARM".CLIENT.U02_STA2_MEAS.ALARMS.CALIBRATION_MISSING_FIX_1_A )
   END_RUNG
   RUNG wire#powerrail
      Contact( "DB16000_OPC_UA_TRIGGER_ALARM".CLIENT.U02_STA2_MEAS.ALARMS.CALIBRATION_MISSING_FIX_1_A )
      I_Contact( "DB2120_MPP_ITC_IPC".RESET_FAULTS )
   END_RUNG wire#w1
   RUNG wire#w2
      Coil( "DB426_ALARMS_WARNINGS".UNIT_02.OTHER."720512" )
   END_RUNG
   // the same network as SCL:
   "DB16000_OPC_UA_TRIGGER_ALARM".CLIENT.U02_STA2_MEAS.ALARMS.CALIBRATION_MISSING_FIX_1_A := ("DB16010_MEASURE_SENSORS_CALIBRATION_STATUS".U02_STA2_MEAS.FIXTURE_1_MISSING OR ("DB16000_OPC_UA_TRIGGER_ALARM".CLIENT.U02_STA2_MEAS.ALARMS.CALIBRATION_MISSING_FIX_1_A AND NOT "DB2120_MPP_ITC_IPC".RESET_FAULTS)) AND NOT "DB2031_CYCLES_GENERAL".CALIBRATION_CYCLE.CYCLE_SELECTED_AUX AND NOT "DB2031_CYCLES_GENERAL".CALIBRATION_CYCLE.CYCLE_SELECTED AND "DB7255_UNIT_02_STA_2_MEAS_ENABLE_DISABLE".ENABLED;
   "DB426_ALARMS_WARNINGS".UNIT_02.OTHER."720512" := "DB16000_OPC_UA_TRIGGER_ALARM".CLIENT.U02_STA2_MEAS.ALARMS.CALIBRATION_MISSING_FIX_1_A;
END_REGION

REGION Network 36: UNIT 02 STATION 2 MISSING CALIBRATION IN FIXTURE 2 ALARM
   RUNG wire#powerrail
      Contact( "DB16010_MEASURE_SENSORS_CALIBRATION_STATUS".U02_STA2_MEAS.FIXTURE_2_MISSING )
      wire#w1
      I_Contact( "DB2031_CYCLES_GENERAL".CALIBRATION_CYCLE.CYCLE_SELECTED_AUX )
      I_Contact( "DB2031_CYCLES_GENERAL".CALIBRATION_CYCLE.CYCLE_SELECTED )
      Contact( "DB7255_UNIT_02_STA_2_MEAS_ENABLE_DISABLE".ENABLED )
      wire#w2
      Coil( "DB16000_OPC_UA_TRIGGER_ALARM".CLIENT.U02_STA2_MEAS.ALARMS.CALIBRATION_MISSING_FIX_2_A )
   END_RUNG
   RUNG wire#powerrail
      Contact( "DB16000_OPC_UA_TRIGGER_ALARM".CLIENT.U02_STA2_MEAS.ALARMS.CALIBRATION_MISSING_FIX_2_A )
      I_Contact( "DB2120_MPP_ITC_IPC".RESET_FAULTS )
   END_RUNG wire#w1
   RUNG wire#w2
      Coil( "DB426_ALARMS_WARNINGS".UNIT_02.OTHER."720513" )
   END_RUNG
   // the same network as SCL:
   "DB16000_OPC_UA_TRIGGER_ALARM".CLIENT.U02_STA2_MEAS.ALARMS.CALIBRATION_MISSING_FIX_2_A := ("DB16010_MEASURE_SENSORS_CALIBRATION_STATUS".U02_STA2_MEAS.FIXTURE_2_MISSING OR ("DB16000_OPC_UA_TRIGGER_ALARM".CLIENT.U02_STA2_MEAS.ALARMS.CALIBRATION_MISSING_FIX_2_A AND NOT "DB2120_MPP_ITC_IPC".RESET_FAULTS)) AND NOT "DB2031_CYCLES_GENERAL".CALIBRATION_CYCLE.CYCLE_SELECTED_AUX AND NOT "DB2031_CYCLES_GENERAL".CALIBRATION_CYCLE.CYCLE_SELECTED AND "DB7255_UNIT_02_STA_2_MEAS_ENABLE_DISABLE".ENABLED;
   "DB426_ALARMS_WARNINGS".UNIT_02.OTHER."720513" := "DB16000_OPC_UA_TRIGGER_ALARM".CLIENT.U02_STA2_MEAS.ALARMS.CALIBRATION_MISSING_FIX_2_A;
END_REGION

REGION Network 37: UNIT 02 STATION 2 MISSING CALIBRATION IN FIXTURE 3 ALARM
   RUNG wire#powerrail
      Contact( "DB16010_MEASURE_SENSORS_CALIBRATION_STATUS".U02_STA2_MEAS.FIXTURE_3_MISSING )
      wire#w1
      I_Contact( "DB2031_CYCLES_GENERAL".CALIBRATION_CYCLE.CYCLE_SELECTED_AUX )
      I_Contact( "DB2031_CYCLES_GENERAL".CALIBRATION_CYCLE.CYCLE_SELECTED )
      Contact( "DB7255_UNIT_02_STA_2_MEAS_ENABLE_DISABLE".ENABLED )
      wire#w2
      Coil( "DB16000_OPC_UA_TRIGGER_ALARM".CLIENT.U02_STA2_MEAS.ALARMS.CALIBRATION_MISSING_FIX_3_A )
   END_RUNG
   RUNG wire#powerrail
      Contact( "DB16000_OPC_UA_TRIGGER_ALARM".CLIENT.U02_STA2_MEAS.ALARMS.CALIBRATION_MISSING_FIX_3_A )
      I_Contact( "DB2120_MPP_ITC_IPC".RESET_FAULTS )
   END_RUNG wire#w1
   RUNG wire#w2
      Coil( "DB426_ALARMS_WARNINGS".UNIT_02.OTHER."720514" )
   END_RUNG
   // the same network as SCL:
   "DB16000_OPC_UA_TRIGGER_ALARM".CLIENT.U02_STA2_MEAS.ALARMS.CALIBRATION_MISSING_FIX_3_A := ("DB16010_MEASURE_SENSORS_CALIBRATION_STATUS".U02_STA2_MEAS.FIXTURE_3_MISSING OR ("DB16000_OPC_UA_TRIGGER_ALARM".CLIENT.U02_STA2_MEAS.ALARMS.CALIBRATION_MISSING_FIX_3_A AND NOT "DB2120_MPP_ITC_IPC".RESET_FAULTS)) AND NOT "DB2031_CYCLES_GENERAL".CALIBRATION_CYCLE.CYCLE_SELECTED_AUX AND NOT "DB2031_CYCLES_GENERAL".CALIBRATION_CYCLE.CYCLE_SELECTED AND "DB7255_UNIT_02_STA_2_MEAS_ENABLE_DISABLE".ENABLED;
   "DB426_ALARMS_WARNINGS".UNIT_02.OTHER."720514" := "DB16000_OPC_UA_TRIGGER_ALARM".CLIENT.U02_STA2_MEAS.ALARMS.CALIBRATION_MISSING_FIX_3_A;
END_REGION

REGION Network 38: UNIT 02 STATION 2 MISSING CALIBRATION IN FIXTURE 4 ALARM
   RUNG wire#powerrail
      Contact( "DB16010_MEASURE_SENSORS_CALIBRATION_STATUS".U02_STA2_MEAS.FIXTURE_4_MISSING )
      wire#w1
      I_Contact( "DB2031_CYCLES_GENERAL".CALIBRATION_CYCLE.CYCLE_SELECTED_AUX )
      I_Contact( "DB2031_CYCLES_GENERAL".CALIBRATION_CYCLE.CYCLE_SELECTED )
      Contact( "DB7255_UNIT_02_STA_2_MEAS_ENABLE_DISABLE".ENABLED )
      wire#w2
      Coil( "DB16000_OPC_UA_TRIGGER_ALARM".CLIENT.U02_STA2_MEAS.ALARMS.CALIBRATION_MISSING_FIX_4_A )
   END_RUNG
   RUNG wire#powerrail
      Contact( "DB16000_OPC_UA_TRIGGER_ALARM".CLIENT.U02_STA2_MEAS.ALARMS.CALIBRATION_MISSING_FIX_4_A )
      I_Contact( "DB2120_MPP_ITC_IPC".RESET_FAULTS )
   END_RUNG wire#w1
   RUNG wire#w2
      Coil( "DB426_ALARMS_WARNINGS".UNIT_02.OTHER."720515" )
   END_RUNG
   // the same network as SCL:
   "DB16000_OPC_UA_TRIGGER_ALARM".CLIENT.U02_STA2_MEAS.ALARMS.CALIBRATION_MISSING_FIX_4_A := ("DB16010_MEASURE_SENSORS_CALIBRATION_STATUS".U02_STA2_MEAS.FIXTURE_4_MISSING OR ("DB16000_OPC_UA_TRIGGER_ALARM".CLIENT.U02_STA2_MEAS.ALARMS.CALIBRATION_MISSING_FIX_4_A AND NOT "DB2120_MPP_ITC_IPC".RESET_FAULTS)) AND NOT "DB2031_CYCLES_GENERAL".CALIBRATION_CYCLE.CYCLE_SELECTED_AUX AND NOT "DB2031_CYCLES_GENERAL".CALIBRATION_CYCLE.CYCLE_SELECTED AND "DB7255_UNIT_02_STA_2_MEAS_ENABLE_DISABLE".ENABLED;
   "DB426_ALARMS_WARNINGS".UNIT_02.OTHER."720515" := "DB16000_OPC_UA_TRIGGER_ALARM".CLIENT.U02_STA2_MEAS.ALARMS.CALIBRATION_MISSING_FIX_4_A;
END_REGION

REGION Network 39: UNIT 02 STATION 2 MEASURING LAST CALIBRATION OUT OF RANGE IN FIXTURE 1 ALARM----------
   RUNG wire#powerrail
      Contact( "DB16010_MEASURE_SENSORS_CALIBRATION_STATUS".U02_STA2_MEAS.FIXTURE_1_MISSING )
      wire#w1
      Contact( "DB7255_UNIT_02_STA_2_MEAS_ENABLE_DISABLE".ENABLED )
      wire#w2
      Coil( "DB16000_OPC_UA_TRIGGER_ALARM".CLIENT.U02_STA2_MEAS.ALARMS.CALIBRATION_OUT_RANGE_FIX_1_A )
   END_RUNG
   RUNG wire#powerrail
      Contact( "DB16000_OPC_UA_TRIGGER_ALARM".CLIENT.U02_STA2_MEAS.ALARMS.CALIBRATION_OUT_RANGE_FIX_1_A )
      I_Contact( "DB2120_MPP_ITC_IPC".RESET_FAULTS )
   END_RUNG wire#w1
   RUNG wire#w2
      Coil( "DB426_ALARMS_WARNINGS".UNIT_02.OTHER."720480" )
   END_RUNG
   // the same network as SCL:
   "DB16000_OPC_UA_TRIGGER_ALARM".CLIENT.U02_STA2_MEAS.ALARMS.CALIBRATION_OUT_RANGE_FIX_1_A := ("DB16010_MEASURE_SENSORS_CALIBRATION_STATUS".U02_STA2_MEAS.FIXTURE_1_MISSING OR ("DB16000_OPC_UA_TRIGGER_ALARM".CLIENT.U02_STA2_MEAS.ALARMS.CALIBRATION_OUT_RANGE_FIX_1_A AND NOT "DB2120_MPP_ITC_IPC".RESET_FAULTS)) AND "DB7255_UNIT_02_STA_2_MEAS_ENABLE_DISABLE".ENABLED;
   "DB426_ALARMS_WARNINGS".UNIT_02.OTHER."720480" := "DB16000_OPC_UA_TRIGGER_ALARM".CLIENT.U02_STA2_MEAS.ALARMS.CALIBRATION_OUT_RANGE_FIX_1_A;
END_REGION

REGION Network 40: UNIT 02 STATION 2 MEASURING LAST CALIBRATION OUT OF RANGE IN FIXTURE 2 ALARM----------
   RUNG wire#powerrail
      Contact( "DB16010_MEASURE_SENSORS_CALIBRATION_STATUS".U02_STA2_MEAS.FIXTURE_2_MISSING )
      wire#w1
      Contact( "DB7255_UNIT_02_STA_2_MEAS_ENABLE_DISABLE".ENABLED )
      wire#w2
      Coil( "DB16000_OPC_UA_TRIGGER_ALARM".CLIENT.U02_STA2_MEAS.ALARMS.CALIBRATION_OUT_RANGE_FIX_2_A )
   END_RUNG
   RUNG wire#powerrail
      Contact( "DB16000_OPC_UA_TRIGGER_ALARM".CLIENT.U02_STA2_MEAS.ALARMS.CALIBRATION_OUT_RANGE_FIX_2_A )
      I_Contact( "DB2120_MPP_ITC_IPC".RESET_FAULTS )
   END_RUNG wire#w1
   RUNG wire#w2
      Coil( "DB426_ALARMS_WARNINGS".UNIT_02.OTHER."720481" )
   END_RUNG
   // the same network as SCL:
   "DB16000_OPC_UA_TRIGGER_ALARM".CLIENT.U02_STA2_MEAS.ALARMS.CALIBRATION_OUT_RANGE_FIX_2_A := ("DB16010_MEASURE_SENSORS_CALIBRATION_STATUS".U02_STA2_MEAS.FIXTURE_2_MISSING OR ("DB16000_OPC_UA_TRIGGER_ALARM".CLIENT.U02_STA2_MEAS.ALARMS.CALIBRATION_OUT_RANGE_FIX_2_A AND NOT "DB2120_MPP_ITC_IPC".RESET_FAULTS)) AND "DB7255_UNIT_02_STA_2_MEAS_ENABLE_DISABLE".ENABLED;
   "DB426_ALARMS_WARNINGS".UNIT_02.OTHER."720481" := "DB16000_OPC_UA_TRIGGER_ALARM".CLIENT.U02_STA2_MEAS.ALARMS.CALIBRATION_OUT_RANGE_FIX_2_A;
END_REGION

REGION Network 41: UNIT 02 STATION 2 MEASURING LAST CALIBRATION OUT OF RANGE IN FIXTURE 3 ALARM----------
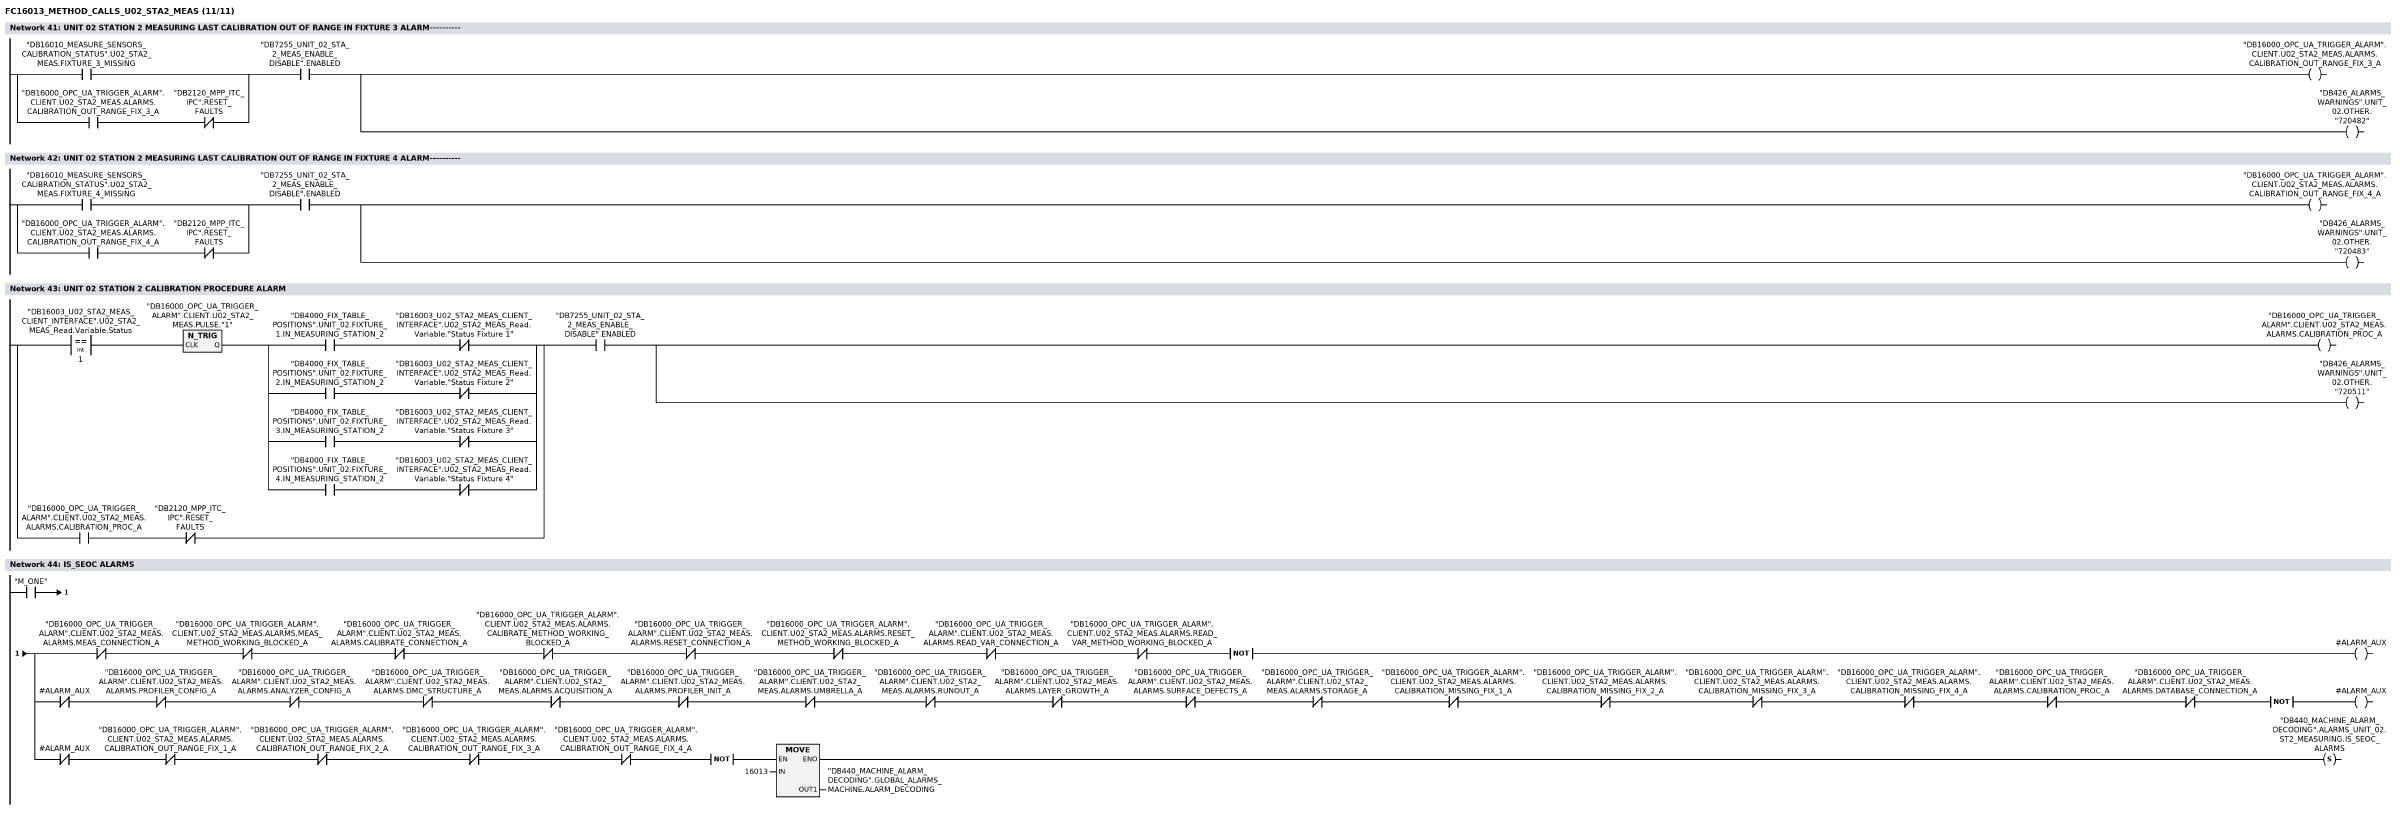
   RUNG wire#powerrail
      Contact( "DB16010_MEASURE_SENSORS_CALIBRATION_STATUS".U02_STA2_MEAS.FIXTURE_3_MISSING )
      wire#w1
      Contact( "DB7255_UNIT_02_STA_2_MEAS_ENABLE_DISABLE".ENABLED )
      wire#w2
      Coil( "DB16000_OPC_UA_TRIGGER_ALARM".CLIENT.U02_STA2_MEAS.ALARMS.CALIBRATION_OUT_RANGE_FIX_3_A )
   END_RUNG
   RUNG wire#powerrail
      Contact( "DB16000_OPC_UA_TRIGGER_ALARM".CLIENT.U02_STA2_MEAS.ALARMS.CALIBRATION_OUT_RANGE_FIX_3_A )
      I_Contact( "DB2120_MPP_ITC_IPC".RESET_FAULTS )
   END_RUNG wire#w1
   RUNG wire#w2
      Coil( "DB426_ALARMS_WARNINGS".UNIT_02.OTHER."720482" )
   END_RUNG
   // the same network as SCL:
   "DB16000_OPC_UA_TRIGGER_ALARM".CLIENT.U02_STA2_MEAS.ALARMS.CALIBRATION_OUT_RANGE_FIX_3_A := ("DB16010_MEASURE_SENSORS_CALIBRATION_STATUS".U02_STA2_MEAS.FIXTURE_3_MISSING OR ("DB16000_OPC_UA_TRIGGER_ALARM".CLIENT.U02_STA2_MEAS.ALARMS.CALIBRATION_OUT_RANGE_FIX_3_A AND NOT "DB2120_MPP_ITC_IPC".RESET_FAULTS)) AND "DB7255_UNIT_02_STA_2_MEAS_ENABLE_DISABLE".ENABLED;
   "DB426_ALARMS_WARNINGS".UNIT_02.OTHER."720482" := "DB16000_OPC_UA_TRIGGER_ALARM".CLIENT.U02_STA2_MEAS.ALARMS.CALIBRATION_OUT_RANGE_FIX_3_A;
END_REGION

REGION Network 42: UNIT 02 STATION 2 MEASURING LAST CALIBRATION OUT OF RANGE IN FIXTURE 4 ALARM----------
   RUNG wire#powerrail
      Contact( "DB16010_MEASURE_SENSORS_CALIBRATION_STATUS".U02_STA2_MEAS.FIXTURE_4_MISSING )
      wire#w1
      Contact( "DB7255_UNIT_02_STA_2_MEAS_ENABLE_DISABLE".ENABLED )
      wire#w2
      Coil( "DB16000_OPC_UA_TRIGGER_ALARM".CLIENT.U02_STA2_MEAS.ALARMS.CALIBRATION_OUT_RANGE_FIX_4_A )
   END_RUNG
   RUNG wire#powerrail
      Contact( "DB16000_OPC_UA_TRIGGER_ALARM".CLIENT.U02_STA2_MEAS.ALARMS.CALIBRATION_OUT_RANGE_FIX_4_A )
      I_Contact( "DB2120_MPP_ITC_IPC".RESET_FAULTS )
   END_RUNG wire#w1
   RUNG wire#w2
      Coil( "DB426_ALARMS_WARNINGS".UNIT_02.OTHER."720483" )
   END_RUNG
   // the same network as SCL:
   "DB16000_OPC_UA_TRIGGER_ALARM".CLIENT.U02_STA2_MEAS.ALARMS.CALIBRATION_OUT_RANGE_FIX_4_A := ("DB16010_MEASURE_SENSORS_CALIBRATION_STATUS".U02_STA2_MEAS.FIXTURE_4_MISSING OR ("DB16000_OPC_UA_TRIGGER_ALARM".CLIENT.U02_STA2_MEAS.ALARMS.CALIBRATION_OUT_RANGE_FIX_4_A AND NOT "DB2120_MPP_ITC_IPC".RESET_FAULTS)) AND "DB7255_UNIT_02_STA_2_MEAS_ENABLE_DISABLE".ENABLED;
   "DB426_ALARMS_WARNINGS".UNIT_02.OTHER."720483" := "DB16000_OPC_UA_TRIGGER_ALARM".CLIENT.U02_STA2_MEAS.ALARMS.CALIBRATION_OUT_RANGE_FIX_4_A;
END_REGION

REGION Network 43: UNIT 02 STATION 2 CALIBRATION PROCEDURE ALARM
   RUNG wire#powerrail
      { S7_Templates := "SrcType := Int" } EQ_Contact(in1 := "DB16003_U02_STA2_MEAS_CLIENT_INTERFACE".U02_STA2_MEAS_Read.Variable.Status, in2 := 1)
      N_Trig( "DB16000_OPC_UA_TRIGGER_ALARM".CLIENT.U02_STA2_MEAS.PULSE."1" )
      wire#w1
      Contact( "DB4000_FIX_TABLE_POSITIONS".UNIT_02.FIXTURE_1.IN_MEASURING_STATION_2 )
      I_Contact( "DB16003_U02_STA2_MEAS_CLIENT_INTERFACE".U02_STA2_MEAS_Read.Variable."Status Fixture 1" )
      wire#w2
      Contact( "DB7255_UNIT_02_STA_2_MEAS_ENABLE_DISABLE".ENABLED )
      wire#w3
      Coil( "DB16000_OPC_UA_TRIGGER_ALARM".CLIENT.U02_STA2_MEAS.ALARMS.CALIBRATION_PROC_A )
   END_RUNG
   RUNG wire#w1
      Contact( "DB4000_FIX_TABLE_POSITIONS".UNIT_02.FIXTURE_2.IN_MEASURING_STATION_2 )
      I_Contact( "DB16003_U02_STA2_MEAS_CLIENT_INTERFACE".U02_STA2_MEAS_Read.Variable."Status Fixture 2" )
   END_RUNG wire#w2
   RUNG wire#w1
      Contact( "DB4000_FIX_TABLE_POSITIONS".UNIT_02.FIXTURE_3.IN_MEASURING_STATION_2 )
      I_Contact( "DB16003_U02_STA2_MEAS_CLIENT_INTERFACE".U02_STA2_MEAS_Read.Variable."Status Fixture 3" )
   END_RUNG wire#w2
   RUNG wire#w1
      Contact( "DB4000_FIX_TABLE_POSITIONS".UNIT_02.FIXTURE_4.IN_MEASURING_STATION_2 )
      I_Contact( "DB16003_U02_STA2_MEAS_CLIENT_INTERFACE".U02_STA2_MEAS_Read.Variable."Status Fixture 4" )
   END_RUNG wire#w2
   RUNG wire#powerrail
      Contact( "DB16000_OPC_UA_TRIGGER_ALARM".CLIENT.U02_STA2_MEAS.ALARMS.CALIBRATION_PROC_A )
      I_Contact( "DB2120_MPP_ITC_IPC".RESET_FAULTS )
   END_RUNG wire#w2
   RUNG wire#w3
      Coil( "DB426_ALARMS_WARNINGS".UNIT_02.OTHER."720511" )
   END_RUNG
   // the same network as SCL:
   #_w1 := "DB16003_U02_STA2_MEAS_CLIENT_INTERFACE".U02_STA2_MEAS_Read.Variable.Status = 1;
   #_w2 := NOT #_w1 AND "DB16000_OPC_UA_TRIGGER_ALARM".CLIENT.U02_STA2_MEAS.PULSE."1";   // falling edge
   "DB16000_OPC_UA_TRIGGER_ALARM".CLIENT.U02_STA2_MEAS.PULSE."1" := #_w1;
   "DB16000_OPC_UA_TRIGGER_ALARM".CLIENT.U02_STA2_MEAS.ALARMS.CALIBRATION_PROC_A := ((#_w2 AND (("DB4000_FIX_TABLE_POSITIONS".UNIT_02.FIXTURE_1.IN_MEASURING_STATION_2 AND NOT "DB16003_U02_STA2_MEAS_CLIENT_INTERFACE".U02_STA2_MEAS_Read.Variable."Status Fixture 1") OR ("DB4000_FIX_TABLE_POSITIONS".UNIT_02.FIXTURE_2.IN_MEASURING_STATION_2 AND NOT "DB16003_U02_STA2_MEAS_CLIENT_INTERFACE".U02_STA2_MEAS_Read.Variable."Status Fixture 2") OR ("DB4000_FIX_TABLE_POSITIONS".UNIT_02.FIXTURE_3.IN_MEASURING_STATION_2 AND NOT "DB16003_U02_STA2_MEAS_CLIENT_INTERFACE".U02_STA2_MEAS_Read.Variable."Status Fixture 3") OR ("DB4000_FIX_TABLE_POSITIONS".UNIT_02.FIXTURE_4.IN_MEASURING_STATION_2 AND NOT "DB16003_U02_STA2_MEAS_CLIENT_INTERFACE".U02_STA2_MEAS_Read.Variable."Status Fixture 4"))) OR ("DB16000_OPC_UA_TRIGGER_ALARM".CLIENT.U02_STA2_MEAS.ALARMS.CALIBRATION_PROC_A AND NOT "DB2120_MPP_ITC_IPC".RESET_FAULTS)) AND "DB7255_UNIT_02_STA_2_MEAS_ENABLE_DISABLE".ENABLED;
   "DB426_ALARMS_WARNINGS".UNIT_02.OTHER."720511" := "DB16000_OPC_UA_TRIGGER_ALARM".CLIENT.U02_STA2_MEAS.ALARMS.CALIBRATION_PROC_A;
END_REGION

REGION Network 44: IS_SEOC ALARMS
   RUNG wire#powerrail
      Contact( "M_ONE" )
      wire#w1
      I_Contact( "DB16000_OPC_UA_TRIGGER_ALARM".CLIENT.U02_STA2_MEAS.ALARMS.MEAS_CONNECTION_A )
      I_Contact( "DB16000_OPC_UA_TRIGGER_ALARM".CLIENT.U02_STA2_MEAS.ALARMS.MEAS_METHOD_WORKING_BLOCKED_A )
      I_Contact( "DB16000_OPC_UA_TRIGGER_ALARM".CLIENT.U02_STA2_MEAS.ALARMS.CALIBRATE_CONNECTION_A )
      I_Contact( "DB16000_OPC_UA_TRIGGER_ALARM".CLIENT.U02_STA2_MEAS.ALARMS.CALIBRATE_METHOD_WORKING_BLOCKED_A )
      I_Contact( "DB16000_OPC_UA_TRIGGER_ALARM".CLIENT.U02_STA2_MEAS.ALARMS.RESET_CONNECTION_A )
      I_Contact( "DB16000_OPC_UA_TRIGGER_ALARM".CLIENT.U02_STA2_MEAS.ALARMS.RESET_METHOD_WORKING_BLOCKED_A )
      I_Contact( "DB16000_OPC_UA_TRIGGER_ALARM".CLIENT.U02_STA2_MEAS.ALARMS.READ_VAR_CONNECTION_A )
      I_Contact( "DB16000_OPC_UA_TRIGGER_ALARM".CLIENT.U02_STA2_MEAS.ALARMS.READ_VAR_METHOD_WORKING_BLOCKED_A )
      Not()
      Coil( #ALARM_AUX )
   END_RUNG
   RUNG wire#w1
      I_Contact( #ALARM_AUX )
      I_Contact( "DB16000_OPC_UA_TRIGGER_ALARM".CLIENT.U02_STA2_MEAS.ALARMS.PROFILER_CONFIG_A )
      I_Contact( "DB16000_OPC_UA_TRIGGER_ALARM".CLIENT.U02_STA2_MEAS.ALARMS.ANALYZER_CONFIG_A )
      I_Contact( "DB16000_OPC_UA_TRIGGER_ALARM".CLIENT.U02_STA2_MEAS.ALARMS.DMC_STRUCTURE_A )
      I_Contact( "DB16000_OPC_UA_TRIGGER_ALARM".CLIENT.U02_STA2_MEAS.ALARMS.ACQUISITION_A )
      I_Contact( "DB16000_OPC_UA_TRIGGER_ALARM".CLIENT.U02_STA2_MEAS.ALARMS.PROFILER_INIT_A )
      I_Contact( "DB16000_OPC_UA_TRIGGER_ALARM".CLIENT.U02_STA2_MEAS.ALARMS.UMBRELLA_A )
      I_Contact( "DB16000_OPC_UA_TRIGGER_ALARM".CLIENT.U02_STA2_MEAS.ALARMS.RUNOUT_A )
      I_Contact( "DB16000_OPC_UA_TRIGGER_ALARM".CLIENT.U02_STA2_MEAS.ALARMS.LAYER_GROWTH_A )
      I_Contact( "DB16000_OPC_UA_TRIGGER_ALARM".CLIENT.U02_STA2_MEAS.ALARMS.SURFACE_DEFECTS_A )
      I_Contact( "DB16000_OPC_UA_TRIGGER_ALARM".CLIENT.U02_STA2_MEAS.ALARMS.STORAGE_A )
      I_Contact( "DB16000_OPC_UA_TRIGGER_ALARM".CLIENT.U02_STA2_MEAS.ALARMS.CALIBRATION_MISSING_FIX_1_A )
      I_Contact( "DB16000_OPC_UA_TRIGGER_ALARM".CLIENT.U02_STA2_MEAS.ALARMS.CALIBRATION_MISSING_FIX_2_A )
      I_Contact( "DB16000_OPC_UA_TRIGGER_ALARM".CLIENT.U02_STA2_MEAS.ALARMS.CALIBRATION_MISSING_FIX_3_A )
      I_Contact( "DB16000_OPC_UA_TRIGGER_ALARM".CLIENT.U02_STA2_MEAS.ALARMS.CALIBRATION_MISSING_FIX_4_A )
      I_Contact( "DB16000_OPC_UA_TRIGGER_ALARM".CLIENT.U02_STA2_MEAS.ALARMS.CALIBRATION_PROC_A )
      I_Contact( "DB16000_OPC_UA_TRIGGER_ALARM".CLIENT.U02_STA2_MEAS.ALARMS.DATABASE_CONNECTION_A )
      Not()
      Coil( #ALARM_AUX )
   END_RUNG
   RUNG wire#w1
      I_Contact( #ALARM_AUX )
      I_Contact( "DB16000_OPC_UA_TRIGGER_ALARM".CLIENT.U02_STA2_MEAS.ALARMS.CALIBRATION_OUT_RANGE_FIX_1_A )
      I_Contact( "DB16000_OPC_UA_TRIGGER_ALARM".CLIENT.U02_STA2_MEAS.ALARMS.CALIBRATION_OUT_RANGE_FIX_2_A )
      I_Contact( "DB16000_OPC_UA_TRIGGER_ALARM".CLIENT.U02_STA2_MEAS.ALARMS.CALIBRATION_OUT_RANGE_FIX_3_A )
      I_Contact( "DB16000_OPC_UA_TRIGGER_ALARM".CLIENT.U02_STA2_MEAS.ALARMS.CALIBRATION_OUT_RANGE_FIX_4_A )
      Not()
      Move(in := 16013, out1 => "DB440_MACHINE_ALARM_DECODING".GLOBAL_ALARMS_MACHINE.ALARM_DECODING)
      S_Coil( "DB440_MACHINE_ALARM_DECODING".ALARMS_UNIT_02.ST2_MEASURING.IS_SEOC_ALARMS )
   END_RUNG
   // the same network as SCL:
   #ALARM_AUX := NOT ("M_ONE" AND NOT "DB16000_OPC_UA_TRIGGER_ALARM".CLIENT.U02_STA2_MEAS.ALARMS.MEAS_CONNECTION_A AND NOT "DB16000_OPC_UA_TRIGGER_ALARM".CLIENT.U02_STA2_MEAS.ALARMS.MEAS_METHOD_WORKING_BLOCKED_A AND NOT "DB16000_OPC_UA_TRIGGER_ALARM".CLIENT.U02_STA2_MEAS.ALARMS.CALIBRATE_CONNECTION_A AND NOT "DB16000_OPC_UA_TRIGGER_ALARM".CLIENT.U02_STA2_MEAS.ALARMS.CALIBRATE_METHOD_WORKING_BLOCKED_A AND NOT "DB16000_OPC_UA_TRIGGER_ALARM".CLIENT.U02_STA2_MEAS.ALARMS.RESET_CONNECTION_A AND NOT "DB16000_OPC_UA_TRIGGER_ALARM".CLIENT.U02_STA2_MEAS.ALARMS.RESET_METHOD_WORKING_BLOCKED_A AND NOT "DB16000_OPC_UA_TRIGGER_ALARM".CLIENT.U02_STA2_MEAS.ALARMS.READ_VAR_CONNECTION_A AND NOT "DB16000_OPC_UA_TRIGGER_ALARM".CLIENT.U02_STA2_MEAS.ALARMS.READ_VAR_METHOD_WORKING_BLOCKED_A);
   #ALARM_AUX := NOT ("M_ONE" AND NOT #ALARM_AUX AND NOT "DB16000_OPC_UA_TRIGGER_ALARM".CLIENT.U02_STA2_MEAS.ALARMS.PROFILER_CONFIG_A AND NOT "DB16000_OPC_UA_TRIGGER_ALARM".CLIENT.U02_STA2_MEAS.ALARMS.ANALYZER_CONFIG_A AND NOT "DB16000_OPC_UA_TRIGGER_ALARM".CLIENT.U02_STA2_MEAS.ALARMS.DMC_STRUCTURE_A AND NOT "DB16000_OPC_UA_TRIGGER_ALARM".CLIENT.U02_STA2_MEAS.ALARMS.ACQUISITION_A AND NOT "DB16000_OPC_UA_TRIGGER_ALARM".CLIENT.U02_STA2_MEAS.ALARMS.PROFILER_INIT_A AND NOT "DB16000_OPC_UA_TRIGGER_ALARM".CLIENT.U02_STA2_MEAS.ALARMS.UMBRELLA_A AND NOT "DB16000_OPC_UA_TRIGGER_ALARM".CLIENT.U02_STA2_MEAS.ALARMS.RUNOUT_A AND NOT "DB16000_OPC_UA_TRIGGER_ALARM".CLIENT.U02_STA2_MEAS.ALARMS.LAYER_GROWTH_A AND NOT "DB16000_OPC_UA_TRIGGER_ALARM".CLIENT.U02_STA2_MEAS.ALARMS.SURFACE_DEFECTS_A AND NOT "DB16000_OPC_UA_TRIGGER_ALARM".CLIENT.U02_STA2_MEAS.ALARMS.STORAGE_A AND NOT "DB16000_OPC_UA_TRIGGER_ALARM".CLIENT.U02_STA2_MEAS.ALARMS.CALIBRATION_MISSING_FIX_1_A AND NOT "DB16000_OPC_UA_TRIGGER_ALARM".CLIENT.U02_STA2_MEAS.ALARMS.CALIBRATION_MISSING_FIX_2_A AND NOT "DB16000_OPC_UA_TRIGGER_ALARM".CLIENT.U02_STA2_MEAS.ALARMS.CALIBRATION_MISSING_FIX_3_A AND NOT "DB16000_OPC_UA_TRIGGER_ALARM".CLIENT.U02_STA2_MEAS.ALARMS.CALIBRATION_MISSING_FIX_4_A AND NOT "DB16000_OPC_UA_TRIGGER_ALARM".CLIENT.U02_STA2_MEAS.ALARMS.CALIBRATION_PROC_A AND NOT "DB16000_OPC_UA_TRIGGER_ALARM".CLIENT.U02_STA2_MEAS.ALARMS.DATABASE_CONNECTION_A);
   IF NOT ("M_ONE" AND NOT #ALARM_AUX AND NOT "DB16000_OPC_UA_TRIGGER_ALARM".CLIENT.U02_STA2_MEAS.ALARMS.CALIBRATION_OUT_RANGE_FIX_1_A AND NOT "DB16000_OPC_UA_TRIGGER_ALARM".CLIENT.U02_STA2_MEAS.ALARMS.CALIBRATION_OUT_RANGE_FIX_2_A AND NOT "DB16000_OPC_UA_TRIGGER_ALARM".CLIENT.U02_STA2_MEAS.ALARMS.CALIBRATION_OUT_RANGE_FIX_3_A AND NOT "DB16000_OPC_UA_TRIGGER_ALARM".CLIENT.U02_STA2_MEAS.ALARMS.CALIBRATION_OUT_RANGE_FIX_4_A) THEN
       "DB440_MACHINE_ALARM_DECODING".GLOBAL_ALARMS_MACHINE.ALARM_DECODING := 16013;
       "DB440_MACHINE_ALARM_DECODING".ALARMS_UNIT_02.ST2_MEASURING.IS_SEOC_ALARMS := TRUE;
   END_IF;
END_REGION
END_FUNCTION
